gfCNCPoint2[12057] = {X 300.6818, Y 64.5076, Z -3.0000, A 0.000, B 0.000, C 0.000 }
gfCNCPoint2[12058] = {X 298.7202, Y 63.1248, Z -3.0000, A 0.000, B 0.000, C 0.000 }
gfCNCPoint2[12059] = {X 298.0340, Y 63.9594, Z -3.0000, A 0.000, B 0.000, C 0.000 }
gfCNCPoint2[12060] = {X 297.2321, Y 64.6835, Z -3.0000, A 0.000, B 0.000, C 0.000 }
gfCNCPoint2[12061] = {X 296.3321, Y 65.2812, Z -3.0000, A 0.000, B 0.000, C 0.000 }
gfCNCPoint2[12062] = {X 296.3321, Y 90.7168, Z -3.0000, A 0.000, B 0.000, C 0.000 }
gfCNCPoint2[12063] = {X 297.3123, Y 91.3793, Z -3.0000, A 0.000, B 0.000, C 0.000 }
gfCNCPoint2[12064] = {X 298.1728, Y 92.1913, Z -3.0000, A 0.000, B 0.000, C 0.000 }
gfCNCPoint2[12065] = {X 298.8912, Y 93.1314, Z -3.0000, A 0.000, B 0.000, C 0.000 }
gfCNCPoint2[12066] = {X 299.4485, Y 94.1751, Z -3.0000, A 0.000, B 0.000, C 0.000 }
gfCNCPoint2[12067] = {X 299.8302, Y 95.2950, Z -3.0000, A 0.000, B 0.000, C 0.000 }
gfCNCPoint2[12068] = {X 308.0994, Y 95.2950, Z -3.0000, A 0.000, B 0.000, C 0.000 }
gfCNCPoint2[12069] = {X 307.0963, Y 93.7116, Z -3.0000, A 0.000, B 0.000, C 0.000 }
gfCNCPoint2[12070] = {X 306.3004, Y 92.0147, Z -3.0000, A 0.000, B 0.000, C 0.000 }
gfCNCPoint2[12071] = {X 305.9924, Y 91.1576, Z -3.0000, A 0.000, B 0.000, C 0.000 }
gfCNCPoint2[12072] = {X 305.7375, Y 90.2832, Z -3.0000, A 0.000, B 0.000, C 0.000 }
gfCNCPoint2[12073] = {X 305.3413, Y 88.4127, Z -3.0000, A 0.000, B 0.000, C 0.000 }
gfCNCPoint2[12074] = {X 305.1069, Y 86.5150, Z -3.0000, A 0.000, B 0.000, C 0.000 }
gfCNCPoint2[12075] = {X 305.0361, Y 84.6043, Z -3.0000, A 0.000, B 0.000, C 0.000 }
gfCNCPoint2[12076] = {X 305.0373, Y 83.2289, Z -3.0000, A 0.000, B 0.000, C 0.000 }
gfCNCPoint2[12077] = {X 305.0373, Y 65.2849, Z -3.0000, A 0.000, B 0.000, C 0.000 }
gfCNCPoint2[12078] = {X 304.1350, Y 64.6870, Z -3.0000, A 0.000, B 0.000, C 0.000 }
gfCNCPoint2[12079] = {X 303.3314, Y 63.9619, Z -3.0000, A 0.000, B 0.000, C 0.000 }
gfCNCPoint2[12080] = {X 302.6441, Y 63.1258, Z -3.0000, A 0.000, B 0.000, C 0.000 }
gfCNCPoint2[12081] = {X 302.0791, Y 62.1784, Z -3.0000, A 0.000, B 0.000, C 0.000 }
gfCNCPoint2[12082] = {X 301.6638, Y 61.1566, Z -3.0000, A 0.000, B 0.000, C 0.000 }
gfCNCPoint2[12083] = {X 301.4076, Y 60.0837, Z -3.0000, A 0.000, B 0.000, C 0.000 }
gfCNCPoint2[12084] = {X 301.3164, Y 58.9845, Z -3.0000, A 0.000, B 0.000, C 0.000 }
gfCNCPoint2[12085] = {X 301.3162, Y 58.0000, Z -3.0000, A 0.000, B 0.000, C 0.000 }
gfCNCPoint2[12086] = {X 301.4018, Y 56.8868, Z -3.0000, A 0.000, B 0.000, C 0.000 }
gfCNCPoint2[12087] = {X 301.6567, Y 55.7997, Z -3.0000, A 0.000, B 0.000, C 0.000 }
gfCNCPoint2[12088] = {X 302.0747, Y 54.7645, Z -3.0000, A 0.000, B 0.000, C 0.000 }
gfCNCPoint2[12089] = {X 302.6462, Y 53.8053, Z -3.0000, A 0.000, B 0.000, C 0.000 }
gfCNCPoint2[12090] = {X 303.3281, Y 52.9755, Z -3.0000, A 0.000, B 0.000, C 0.000 }
gfCNCPoint2[12091] = {X 304.1247, Y 52.2551, Z -3.0000, A 0.000, B 0.000, C 0.000 }
gfCNCPoint2[12092] = {X 305.0187, Y 51.6597, Z -3.0000, A 0.000, B 0.000, C 0.000 }
gfCNCPoint2[12093] = {X 306.1514, Y 51.1428, Z -3.0000, A 0.000, B 0.000, C 0.000 }
gfCNCPoint2[12094] = {X 307.3557, Y 50.8265, Z -3.0000, A 0.000, B 0.000, C 0.000 }
gfCNCPoint2[12095] = {X 308.5962, Y 50.7200, Z -3.0000, A 0.000, B 0.000, C 0.000 }
gfCNCPoint2[12096] = {X 324.3107, Y 50.7200, Z -3.0000, A 0.000, B 0.000, C 0.000 }
gfCNCPoint2[12097] = {X 325.2469, Y 50.7804, Z -3.0000, A 0.000, B 0.000, C 0.000 }
gfCNCPoint2[12098] = {X 326.1675, Y 50.9608, Z -3.0000, A 0.000, B 0.000, C 0.000 }
gfCNCPoint2[12099] = {X 326.5260, Y 51.0653, Z -3.0000, A 0.000, B 0.000, C 0.000 }
gfCNCPoint2[12100] = {X 326.8787, Y 51.1880, Z -3.0000, A 0.000, B 0.000, C 0.000 }
gfCNCPoint2[12101] = {X 327.4520, Y 51.4326, Z -3.0000, A 0.000, B 0.000, C 0.000 }
gfCNCPoint2[12102] = {X 328.0023, Y 51.7254, Z -3.0000, A 0.000, B 0.000, C 0.000 }
gfCNCPoint2[12103] = {X 328.5421, Y 52.0760, Z -3.0000, A 0.000, B 0.000, C 0.000 }
gfCNCPoint2[12104] = {X 329.0488, Y 52.4729, Z -3.0000, A 0.000, B 0.000, C 0.000 }
gfCNCPoint2[12105] = {X 329.9268, Y 53.3678, Z -3.0000, A 0.000, B 0.000, C 0.000 }
gfCNCPoint2[12106] = {X 330.6383, Y 54.4000, Z -3.0000, A 0.000, B 0.000, C 0.000 }
gfCNCPoint2[12107] = {X 331.1621, Y 55.5390, Z -3.0000, A 0.000, B 0.000, C 0.000 }
gfCNCPoint2[12108] = {X 331.4827, Y 56.7510, Z -3.0000, A 0.000, B 0.000, C 0.000 }
gfCNCPoint2[12109] = {X 331.5907, Y 58.0000, Z -3.0000, A 0.000, B 0.000, C 0.000 }
gfCNCPoint2[12110] = {X 331.5907, Y 58.9400, Z -3.0000, A 0.000, B 0.000, C 0.000 }
gfCNCPoint2[12111] = {X 331.4731, Y 60.2169, Z -3.0000, A 0.000, B 0.000, C 0.000 }
gfCNCPoint2[12112] = {X 331.1345, Y 61.4536, Z -3.0000, A 0.000, B 0.000, C 0.000 }
gfCNCPoint2[12113] = {X 330.5852, Y 62.6123, Z -3.0000, A 0.000, B 0.000, C 0.000 }
gfCNCPoint2[12114] = {X 329.8422, Y 63.6573, Z -3.0000, A 0.000, B 0.000, C 0.000 }
gfCNCPoint2[12115] = {X 328.9282, Y 64.5567, Z -3.0000, A 0.000, B 0.000, C 0.000 }
gfCNCPoint2[12116] = {X 327.8712, Y 65.2827, Z -3.0000, A 0.000, B 0.000, C 0.000 }
gfCNCPoint2[12117] = {X 327.8726, Y 83.2150, Z -3.0000, A 0.000, B 0.000, C 0.000 }
gfCNCPoint2[12118] = {X 327.8860, Y 84.5922, Z -3.0000, A 0.000, B 0.000, C 0.000 }
gfCNCPoint2[12119] = {X 327.8954, Y 84.9546, Z -3.0000, A 0.000, B 0.000, C 0.000 }
gfCNCPoint2[12120] = {X 327.9223, Y 85.3160, Z -3.0000, A 0.000, B 0.000, C 0.000 }
gfCNCPoint2[12121] = {X 328.8635, Y 85.6736, Z -3.0000, A 0.000, B 0.000, C 0.000 }
gfCNCPoint2[12122] = {X 329.8331, Y 85.9449, Z -3.0000, A 0.000, B 0.000, C 0.000 }
gfCNCPoint2[12123] = {X 332.7072, Y 86.5208, Z -3.0000, A 0.000, B 0.000, C 0.000 }
gfCNCPoint2[12124] = {X 335.6155, Y 86.8875, Z -3.0000, A 0.000, B 0.000, C 0.000 }
gfCNCPoint2[12125] = {X 339.6624, Y 87.2011, Z -3.0000, A 0.000, B 0.000, C 0.000 }
gfCNCPoint2[12126] = {X 343.7177, Y 87.3767, Z -3.0000, A 0.000, B 0.000, C 0.000 }
gfCNCPoint2[12127] = {X 347.7766, Y 87.4140, Z -3.0000, A 0.000, B 0.000, C 0.000 }
gfCNCPoint2[12128] = {X 352.0642, Y 87.3773, Z -3.0000, A 0.000, B 0.000, C 0.000 }
gfCNCPoint2[12129] = {X 356.3477, Y 87.1860, Z -3.0000, A 0.000, B 0.000, C 0.000 }
gfCNCPoint2[12130] = {X 360.6216, Y 86.8405, Z -3.0000, A 0.000, B 0.000, C 0.000 }
gfCNCPoint2[12131] = {X 362.7646, Y 86.5743, Z -3.0000, A 0.000, B 0.000, C 0.000 }
gfCNCPoint2[12132] = {X 364.8876, Y 86.1795, Z -3.0000, A 0.000, B 0.000, C 0.000 }
gfCNCPoint2[12133] = {X 366.9831, Y 85.6575, Z -3.0000, A 0.000, B 0.000, C 0.000 }
gfCNCPoint2[12134] = {X 367.4432, Y 85.5111, Z -3.0000, A 0.000, B 0.000, C 0.000 }
gfCNCPoint2[12135] = {X 367.8895, Y 85.3269, Z -3.0000, A 0.000, B 0.000, C 0.000 }
gfCNCPoint2[12136] = {X 367.9430, Y 84.5784, Z -3.0000, A 0.000, B 0.000, C 0.000 }
gfCNCPoint2[12137] = {X 367.9608, Y 83.8282, Z -3.0000, A 0.000, B 0.000, C 0.000 }
gfCNCPoint2[12138] = {X 367.9593, Y 65.2843, Z -3.0000, A 0.000, B 0.000, C 0.000 }
gfCNCPoint2[12139] = {X 366.9053, Y 64.5652, Z -3.0000, A 0.000, B 0.000, C 0.000 }
gfCNCPoint2[12140] = {X 365.9931, Y 63.6732, Z -3.0000, A 0.000, B 0.000, C 0.000 }
gfCNCPoint2[12141] = {X 365.2505, Y 62.6356, Z -3.0000, A 0.000, B 0.000, C 0.000 }
gfCNCPoint2[12142] = {X 364.7006, Y 61.4843, Z -3.0000, A 0.000, B 0.000, C 0.000 }
gfCNCPoint2[12143] = {X 364.3601, Y 60.2547, Z -3.0000, A 0.000, B 0.000, C 0.000 }
gfCNCPoint2[12144] = {X 364.2395, Y 58.9845, Z -3.0000, A 0.000, B 0.000, C 0.000 }
gfCNCPoint2[12145] = {X 364.2393, Y 58.0000, Z -3.0000, A 0.000, B 0.000, C 0.000 }
gfCNCPoint2[12146] = {X 364.3499, Y 56.7358, Z -3.0000, A 0.000, B 0.000, C 0.000 }
gfCNCPoint2[12147] = {X 364.6783, Y 55.5101, Z -3.0000, A 0.000, B 0.000, C 0.000 }
gfCNCPoint2[12148] = {X 365.2146, Y 54.3600, Z -3.0000, A 0.000, B 0.000, C 0.000 }
gfCNCPoint2[12149] = {X 365.9425, Y 53.3205, Z -3.0000, A 0.000, B 0.000, C 0.000 }
gfCNCPoint2[12150] = {X 366.8398, Y 52.4232, Z -3.0000, A 0.000, B 0.000, C 0.000 }
gfCNCPoint2[12151] = {X 367.8793, Y 51.6953, Z -3.0000, A 0.000, B 0.000, C 0.000 }
gfCNCPoint2[12152] = {X 369.0294, Y 51.1590, Z -3.0000, A 0.000, B 0.000, C 0.000 }
gfCNCPoint2[12153] = {X 370.2551, Y 50.8306, Z -3.0000, A 0.000, B 0.000, C 0.000 }
gfCNCPoint2[12154] = {X 371.5193, Y 50.7200, Z -3.0000, A 0.000, B 0.000, C 0.000 }
gfCNCPoint2[12155] = {X 388.0597, Y 50.7200, Z -3.0000, A 0.000, B 0.000, C 0.000 }
gfCNCPoint2[12156] = {X 389.2271, Y 50.8142, Z -3.0000, A 0.000, B 0.000, C 0.000 }
gfCNCPoint2[12157] = {X 390.3643, Y 51.0944, Z -3.0000, A 0.000, B 0.000, C 0.000 }
gfCNCPoint2[12158] = {X 391.4418, Y 51.5533, Z -3.0000, A 0.000, B 0.000, C 0.000 }
gfCNCPoint2[12159] = {X 392.4319, Y 52.1791, Z -3.0000, A 0.000, B 0.000, C 0.000 }
gfCNCPoint2[12160] = {X 393.3087, Y 52.9556, Z -3.0000, A 0.000, B 0.000, C 0.000 }
gfCNCPoint2[12161] = {X 394.1855, Y 52.1791, Z -3.0000, A 0.000, B 0.000, C 0.000 }
gfCNCPoint2[12162] = {X 395.1756, Y 51.5533, Z -3.0000, A 0.000, B 0.000, C 0.000 }
gfCNCPoint2[12163] = {X 396.2531, Y 51.0944, Z -3.0000, A 0.000, B 0.000, C 0.000 }
gfCNCPoint2[12164] = {X 397.3903, Y 50.8142, Z -3.0000, A 0.000, B 0.000, C 0.000 }
gfCNCPoint2[12165] = {X 398.5577, Y 50.7200, Z -3.0000, A 0.000, B 0.000, C 0.000 }
gfCNCPoint2[12166] = {X 419.4886, Y 50.7200, Z -3.0000, A 0.000, B 0.000, C 0.000 }
gfCNCPoint2[12167] = {X 420.6740, Y 50.8172, Z -3.0000, A 0.000, B 0.000, C 0.000 }
gfCNCPoint2[12168] = {X 421.8278, Y 51.1060, Z -3.0000, A 0.000, B 0.000, C 0.000 }
gfCNCPoint2[12169] = {X 422.9191, Y 51.5790, Z -3.0000, A 0.000, B 0.000, C 0.000 }
gfCNCPoint2[12170] = {X 423.9189, Y 52.2233, Z -3.0000, A 0.000, B 0.000, C 0.000 }
gfCNCPoint2[12171] = {X 424.8004, Y 53.0217, Z -3.0000, A 0.000, B 0.000, C 0.000 }
gfCNCPoint2[12172] = {X 425.5401, Y 53.9531, Z -3.0000, A 0.000, B 0.000, C 0.000 }
gfCNCPoint2[12173] = {X 426.1183, Y 54.9925, Z -3.0000, A 0.000, B 0.000, C 0.000 }
gfCNCPoint2[12174] = {X 426.5196, Y 56.1122, Z -3.0000, A 0.000, B 0.000, C 0.000 }
gfCNCPoint2[12175] = {X 430.7007, Y 57.7417, Z -3.0000, A 0.000, B 0.000, C 0.000 }
gfCNCPoint2[12176] = {X 454.9001, Y 67.3428, Z -3.0000, A 0.000, B 0.000, C 0.000 }
gfCNCPoint2[12177] = {X 454.8999, Y 65.2844, Z -3.0000, A 0.000, B 0.000, C 0.000 }
gfCNCPoint2[12178] = {X 453.8924, Y 64.6032, Z -3.0000, A 0.000, B 0.000, C 0.000 }
gfCNCPoint2[12179] = {X 453.0124, Y 63.7638, Z -3.0000, A 0.000, B 0.000, C 0.000 }
gfCNCPoint2[12180] = {X 452.2844, Y 62.7896, Z -3.0000, A 0.000, B 0.000, C 0.000 }
gfCNCPoint2[12181] = {X 451.7287, Y 61.7078, Z -3.0000, A 0.000, B 0.000, C 0.000 }
gfCNCPoint2[12182] = {X 451.4297, Y 60.8260, Z -3.0000, A 0.000, B 0.000, C 0.000 }
gfCNCPoint2[12183] = {X 451.2457, Y 59.9132, Z -3.0000, A 0.000, B 0.000, C 0.000 }
gfCNCPoint2[12184] = {X 451.1798, Y 58.9845, Z -3.0000, A 0.000, B 0.000, C 0.000 }
gfCNCPoint2[12185] = {X 451.1796, Y 58.0000, Z -3.0000, A 0.000, B 0.000, C 0.000 }
gfCNCPoint2[12186] = {X 451.2795, Y 56.7981, Z -3.0000, A 0.000, B 0.000, C 0.000 }
gfCNCPoint2[12187] = {X 451.5765, Y 55.6291, Z -3.0000, A 0.000, B 0.000, C 0.000 }
gfCNCPoint2[12188] = {X 452.0624, Y 54.5253, Z -3.0000, A 0.000, B 0.000, C 0.000 }
gfCNCPoint2[12189] = {X 452.7238, Y 53.5168, Z -3.0000, A 0.000, B 0.000, C 0.000 }
gfCNCPoint2[12190] = {X 453.5427, Y 52.6313, Z -3.0000, A 0.000, B 0.000, C 0.000 }
gfCNCPoint2[12191] = {X 454.4966, Y 51.8932, Z -3.0000, A 0.000, B 0.000, C 0.000 }
gfCNCPoint2[12192] = {X 455.4133, Y 51.3880, Z -3.0000, A 0.000, B 0.000, C 0.000 }
gfCNCPoint2[12193] = {X 456.3931, Y 51.0195, Z -3.0000, A 0.000, B 0.000, C 0.000 }
gfCNCPoint2[12194] = {X 457.4155, Y 50.7953, Z -3.0000, A 0.000, B 0.000, C 0.000 }
gfCNCPoint2[12195] = {X 458.4596, Y 50.7200, Z -3.0000, A 0.000, B 0.000, C 0.000 }
gfCNCPoint2[12196] = {X 475.0000, Y 50.7200, Z -3.0000, A 0.000, B 0.000, C 0.000 }
gfCNCPoint2[12197] = {X 476.0441, Y 50.7953, Z -3.0000, A 0.000, B 0.000, C 0.000 }
gfCNCPoint2[12198] = {X 477.0665, Y 51.0195, Z -3.0000, A 0.000, B 0.000, C 0.000 }
gfCNCPoint2[12199] = {X 478.0463, Y 51.3880, Z -3.0000, A 0.000, B 0.000, C 0.000 }
gfCNCPoint2[12200] = {X 478.9630, Y 51.8932, Z -3.0000, A 0.000, B 0.000, C 0.000 }
gfCNCPoint2[12201] = {X 479.9169, Y 52.6313, Z -3.0000, A 0.000, B 0.000, C 0.000 }
gfCNCPoint2[12202] = {X 480.7358, Y 53.5168, Z -3.0000, A 0.000, B 0.000, C 0.000 }
gfCNCPoint2[12203] = {X 481.3972, Y 54.5253, Z -3.0000, A 0.000, B 0.000, C 0.000 }
gfCNCPoint2[12204] = {X 481.8831, Y 55.6291, Z -3.0000, A 0.000, B 0.000, C 0.000 }
gfCNCPoint2[12205] = {X 482.1801, Y 56.7981, Z -3.0000, A 0.000, B 0.000, C 0.000 }
gfCNCPoint2[12206] = {X 482.2800, Y 58.0000, Z -3.0000, A 0.000, B 0.000, C 0.000 }
gfCNCPoint2[12207] = {X 482.2798, Y 58.9942, Z -3.0000, A 0.000, B 0.000, C 0.000 }
gfCNCPoint2[12208] = {X 482.1577, Y 60.2627, Z -3.0000, A 0.000, B 0.000, C 0.000 }
gfCNCPoint2[12209] = {X 481.8164, Y 61.4904, Z -3.0000, A 0.000, B 0.000, C 0.000 }
gfCNCPoint2[12210] = {X 481.2662, Y 62.6399, Z -3.0000, A 0.000, B 0.000, C 0.000 }
gfCNCPoint2[12211] = {X 480.5240, Y 63.6758, Z -3.0000, A 0.000, B 0.000, C 0.000 }
gfCNCPoint2[12212] = {X 479.6125, Y 64.5664, Z -3.0000, A 0.000, B 0.000, C 0.000 }
gfCNCPoint2[12213] = {X 478.5597, Y 65.2844, Z -3.0000, A 0.000, B 0.000, C 0.000 }
gfCNCPoint2[12214] = {X 478.5601, Y 90.7248, Z -3.0000, A 0.000, B 0.000, C 0.000 }
gfCNCPoint2[12215] = {X 479.5426, Y 91.3833, Z -3.0000, A 0.000, B 0.000, C 0.000 }
gfCNCPoint2[12216] = {X 480.4051, Y 92.1928, Z -3.0000, A 0.000, B 0.000, C 0.000 }
gfCNCPoint2[12217] = {X 481.1245, Y 93.1317, Z -3.0000, A 0.000, B 0.000, C 0.000 }
gfCNCPoint2[12218] = {X 481.6818, Y 94.1750, Z -3.0000, A 0.000, B 0.000, C 0.000 }
gfCNCPoint2[12219] = {X 482.0621, Y 95.2950, Z -3.0000, A 0.000, B 0.000, C 0.000 }
gfCNCPoint2[12220] = {X 507.6818, Y 95.2950, Z -3.0000, A 0.000, B 0.000, C 0.000 }
gfCNCPoint2[12221] = {X 507.6818, Y 97.6950, Z -3.0000, A 0.000, B 0.000, C 0.000 }
gfCNCPoint2[12222] = {X 597.6965, Y 97.6950, Z -3.0000, A 0.000, B 0.000, C 0.000 }
gfCNCPoint2[12223] = {X 597.6965, Y 51.8000, Z -3.0000, A 0.000, B 0.000, C 0.000 }
gfCNCPoint2[12224] = {X 593.5565, Y 51.8000, Z -3.0000, A 0.000, B 0.000, C 0.000 }
gfCNCPoint2[12225] = {X 592.3428, Y 51.6908, Z -3.0000, A 0.000, B 0.000, C 0.000 }
gfCNCPoint2[12226] = {X 591.1680, Y 51.3667, Z -3.0000, A 0.000, B 0.000, C 0.000 }
gfCNCPoint2[12227] = {X 590.0699, Y 50.8381, Z -3.0000, A 0.000, B 0.000, C 0.000 }
gfCNCPoint2[12228] = {X 589.0838, Y 50.1220, Z -3.0000, A 0.000, B 0.000, C 0.000 }
gfCNCPoint2[12229] = {X 588.4736, Y 49.5171, Z -3.0000, A 0.000, B 0.000, C 0.000 }
gfCNCPoint2[12230] = {X 587.9446, Y 48.8401, Z -3.0000, A 0.000, B 0.000, C 0.000 }
gfCNCPoint2[12231] = {X 587.5052, Y 48.1018, Z -3.0000, A 0.000, B 0.000, C 0.000 }
gfCNCPoint2[12232] = {X 587.0658, Y 48.8401, Z -3.0000, A 0.000, B 0.000, C 0.000 }
gfCNCPoint2[12233] = {X 586.5368, Y 49.5171, Z -3.0000, A 0.000, B 0.000, C 0.000 }
gfCNCPoint2[12234] = {X 585.9266, Y 50.1220, Z -3.0000, A 0.000, B 0.000, C 0.000 }
gfCNCPoint2[12235] = {X 585.1803, Y 50.6880, Z -3.0000, A 0.000, B 0.000, C 0.000 }
gfCNCPoint2[12236] = {X 584.3634, Y 51.1461, Z -3.0000, A 0.000, B 0.000, C 0.000 }
gfCNCPoint2[12237] = {X 583.3013, Y 51.5442, Z -3.0000, A 0.000, B 0.000, C 0.000 }
gfCNCPoint2[12238] = {X 582.1877, Y 51.7603, Z -3.0000, A 0.000, B 0.000, C 0.000 }
gfCNCPoint2[12239] = {X 581.0538, Y 51.7882, Z -3.0000, A 0.000, B 0.000, C 0.000 }
gfCNCPoint2[12240] = {X 579.9310, Y 51.6273, Z -3.0000, A 0.000, B 0.000, C 0.000 }
gfCNCPoint2[12241] = {X 578.8505, Y 51.2819, Z -3.0000, A 0.000, B 0.000, C 0.000 }
gfCNCPoint2[12242] = {X 577.8425, Y 50.7618, Z -3.0000, A 0.000, B 0.000, C 0.000 }
gfCNCPoint2[12243] = {X 576.9350, Y 50.0813, Z -3.0000, A 0.000, B 0.000, C 0.000 }
gfCNCPoint2[12244] = {X 576.3133, Y 49.4513, Z -3.0000, A 0.000, B 0.000, C 0.000 }
gfCNCPoint2[12245] = {X 575.7786, Y 48.7459, Z -3.0000, A 0.000, B 0.000, C 0.000 }
gfCNCPoint2[12246] = {X 575.3401, Y 47.9770, Z -3.0000, A 0.000, B 0.000, C 0.000 }
gfCNCPoint2[12247] = {X 574.7637, Y 48.9470, Z -3.0000, A 0.000, B 0.000, C 0.000 }
gfCNCPoint2[12248] = {X 574.0348, Y 49.8083, Z -3.0000, A 0.000, B 0.000, C 0.000 }
gfCNCPoint2[12249] = {X 573.8920, Y 49.9470, Z -3.0000, A 0.000, B 0.000, C 0.000 }
gfCNCPoint2[12250] = {X 573.7453, Y 50.0813, Z -3.0000, A 0.000, B 0.000, C 0.000 }
gfCNCPoint2[12251] = {X 572.7526, Y 50.8143, Z -3.0000, A 0.000, B 0.000, C 0.000 }
gfCNCPoint2[12252] = {X 571.6437, Y 51.3558, Z -3.0000, A 0.000, B 0.000, C 0.000 }
gfCNCPoint2[12253] = {X 570.4553, Y 51.6880, Z -3.0000, A 0.000, B 0.000, C 0.000 }
gfCNCPoint2[12254] = {X 569.2264, Y 51.8000, Z -3.0000, A 0.000, B 0.000, C 0.000 }
gfCNCPoint2[12255] = {X 562.4443, Y 51.8000, Z -3.0000, A 0.000, B 0.000, C 0.000 }
gfCNCPoint2[12256] = {X 561.2635, Y 51.6967, Z -3.0000, A 0.000, B 0.000, C 0.000 }
gfCNCPoint2[12257] = {X 560.1186, Y 51.3899, Z -3.0000, A 0.000, B 0.000, C 0.000 }
gfCNCPoint2[12258] = {X 559.0443, Y 50.8890, Z -3.0000, A 0.000, B 0.000, C 0.000 }
gfCNCPoint2[12259] = {X 558.0733, Y 50.2091, Z -3.0000, A 0.000, B 0.000, C 0.000 }
gfCNCPoint2[12260] = {X 557.2352, Y 49.3710, Z -3.0000, A 0.000, B 0.000, C 0.000 }
gfCNCPoint2[12261] = {X 556.5553, Y 48.4000, Z -3.0000, A 0.000, B 0.000, C 0.000 }
gfCNCPoint2[12262] = {X 556.0544, Y 47.3257, Z -3.0000, A 0.000, B 0.000, C 0.000 }
gfCNCPoint2[12263] = {X 555.7476, Y 46.1808, Z -3.0000, A 0.000, B 0.000, C 0.000 }
gfCNCPoint2[12264] = {X 555.6443, Y 45.0000, Z -3.0000, A 0.000, B 0.000, C 0.000 }
gfCNCPoint2[12265] = {X 555.6443, Y 44.0663, Z -3.0000, A 0.000, B 0.000, C 0.000 }
gfCNCPoint2[12266] = {X 555.7457, Y 42.9115, Z -3.0000, A 0.000, B 0.000, C 0.000 }
gfCNCPoint2[12267] = {X 556.0407, Y 41.7905, Z -3.0000, A 0.000, B 0.000, C 0.000 }
gfCNCPoint2[12268] = {X 556.5208, Y 40.7354, Z -3.0000, A 0.000, B 0.000, C 0.000 }
gfCNCPoint2[12269] = {X 557.1724, Y 39.7767, Z -3.0000, A 0.000, B 0.000, C 0.000 }
gfCNCPoint2[12270] = {X 557.1724, Y 10.2290, Z -3.0000, A 0.000, B 0.000, C 0.000 }
gfCNCPoint2[12271] = {X 556.5260, Y 9.2828, Z -3.0000, A 0.000, B 0.000, C 0.000 }
gfCNCPoint2[12272] = {X 556.0477, Y 8.2414, Z -3.0000, A 0.000, B 0.000, C 0.000 }
gfCNCPoint2[12273] = {X 555.7511, Y 7.1345, Z -3.0000, A 0.000, B 0.000, C 0.000 }
gfCNCPoint2[12274] = {X 555.6446, Y 5.9935, Z -3.0000, A 0.000, B 0.000, C 0.000 }
gfCNCPoint2[12275] = {X 555.6443, Y 5.0000, Z -3.0000, A 0.000, B 0.000, C 0.000 }
gfCNCPoint2[12276] = {X 555.6452, Y 4.8910, Z -3.0000, A 0.000, B 0.000, C 0.000 }
gfCNCPoint2[12277] = {X 555.6478, Y 4.7820, Z -3.0000, A 0.000, B 0.000, C 0.000 }
gfCNCPoint2[12278] = {X 555.8079, Y 3.5175, Z -3.0000, A 0.000, B 0.000, C 0.000 }
gfCNCPoint2[12279] = {X 556.2011, Y 2.3050, Z -3.0000, A 0.000, B 0.000, C 0.000 }
gfCNCPoint2[12280] = {X 358.2581, Y 2.3050, Z -3.0000, A 0.000, B 0.000, C 0.000 }
gfCNCPoint2[12281] = {X 360.1196, Y 3.4747, Z -3.0000, A 0.000, B 0.000, C 0.000 }
gfCNCPoint2[12282] = {X 361.8525, Y 4.8276, Z -3.0000, A 0.000, B 0.000, C 0.000 }
gfCNCPoint2[12283] = {X 363.4387, Y 6.3498, Z -3.0000, A 0.000, B 0.000, C 0.000 }
gfCNCPoint2[12284] = {X 363.7843, Y 6.7258, Z -3.0000, A 0.000, B 0.000, C 0.000 }
gfCNCPoint2[12285] = {X 364.1208, Y 7.1099, Z -3.0000, A 0.000, B 0.000, C 0.000 }
gfCNCPoint2[12286] = {X 365.6213, Y 9.0462, Z -3.0000, A 0.000, B 0.000, C 0.000 }
gfCNCPoint2[12287] = {X 366.9272, Y 11.1187, Z -3.0000, A 0.000, B 0.000, C 0.000 }
gfCNCPoint2[12288] = {X 368.0265, Y 13.3079, Z -3.0000, A 0.000, B 0.000, C 0.000 }
gfCNCPoint2[12289] = {X 368.9087, Y 15.5932, Z -3.0000, A 0.000, B 0.000, C 0.000 }
gfCNCPoint2[12290] = {X 369.5655, Y 17.9532, Z -3.0000, A 0.000, B 0.000, C 0.000 }
gfCNCPoint2[12291] = {X 370.0551, Y 20.6344, Z -3.0000, A 0.000, B 0.000, C 0.000 }
gfCNCPoint2[12292] = {X 370.3162, Y 23.3475, Z -3.0000, A 0.000, B 0.000, C 0.000 }
gfCNCPoint2[12293] = {X 370.3467, Y 26.0729, Z -3.0000, A 0.000, B 0.000, C 0.000 }
gfCNCPoint2[12294] = {X 370.1465, Y 28.7912, Z -3.0000, A 0.000, B 0.000, C 0.000 }
gfCNCPoint2[12295] = {X 369.7171, Y 31.4827, Z -3.0000, A 0.000, B 0.000, C 0.000 }
gfCNCPoint2[12296] = {X 369.1813, Y 33.6350, Z -3.0000, A 0.000, B 0.000, C 0.000 }
gfCNCPoint2[12297] = {X 368.4574, Y 35.7315, Z -3.0000, A 0.000, B 0.000, C 0.000 }
gfCNCPoint2[12298] = {X 367.5511, Y 37.7559, Z -3.0000, A 0.000, B 0.000, C 0.000 }
gfCNCPoint2[12299] = {X 366.4695, Y 39.6923, Z -3.0000, A 0.000, B 0.000, C 0.000 }
gfCNCPoint2[12300] = {X 365.2210, Y 41.5255, Z -3.0000, A 0.000, B 0.000, C 0.000 }
gfCNCPoint2[12301] = {X 363.9635, Y 43.0750, Z -3.0000, A 0.000, B 0.000, C 0.000 }
gfCNCPoint2[12302] = {X 362.5750, Y 44.5082, Z -3.0000, A 0.000, B 0.000, C 0.000 }
gfCNCPoint2[12303] = {X 361.0663, Y 45.8143, Z -3.0000, A 0.000, B 0.000, C 0.000 }
gfCNCPoint2[12304] = {X 359.4488, Y 46.9830, Z -3.0000, A 0.000, B 0.000, C 0.000 }
gfCNCPoint2[12305] = {X 357.7352, Y 48.0055, Z -3.0000, A 0.000, B 0.000, C 0.000 }
gfCNCPoint2[12306] = {X 355.7254, Y 48.9198, Z -3.0000, A 0.000, B 0.000, C 0.000 }
gfCNCPoint2[12307] = {X 353.6378, Y 49.6388, Z -3.0000, A 0.000, B 0.000, C 0.000 }
gfCNCPoint2[12308] = {X 351.4913, Y 50.1561, Z -3.0000, A 0.000, B 0.000, C 0.000 }
gfCNCPoint2[12309] = {X 349.3053, Y 50.4668, Z -3.0000, A 0.000, B 0.000, C 0.000 }
gfCNCPoint2[12310] = {X 347.0997, Y 50.5683, Z -3.0000, A 0.000, B 0.000, C 0.000 }
gfCNCPoint2[12311] = {X 344.9865, Y 50.5320, Z -3.0000, A 0.000, B 0.000, C 0.000 }
gfCNCPoint2[12312] = {X 342.8843, Y 50.3128, Z -3.0000, A 0.000, B 0.000, C 0.000 }
gfCNCPoint2[12313] = {X 340.8090, Y 49.9122, Z -3.0000, A 0.000, B 0.000, C 0.000 }
gfCNCPoint2[12314] = {X 338.7763, Y 49.3332, Z -3.0000, A 0.000, B 0.000, C 0.000 }
gfCNCPoint2[12315] = {X 336.8014, Y 48.5803, Z -3.0000, A 0.000, B 0.000, C 0.000 }
gfCNCPoint2[12316] = {X 334.8991, Y 47.6591, Z -3.0000, A 0.000, B 0.000, C 0.000 }
gfCNCPoint2[12317] = {X 333.3420, Y 46.7029, Z -3.0000, A 0.000, B 0.000, C 0.000 }
gfCNCPoint2[12318] = {X 331.8608, Y 45.6328, Z -3.0000, A 0.000, B 0.000, C 0.000 }
gfCNCPoint2[12319] = {X 330.4638, Y 44.4550, Z -3.0000, A 0.000, B 0.000, C 0.000 }
gfCNCPoint2[12320] = {X 329.4666, Y 44.4079, Z -3.0000, A 0.000, B 0.000, C 0.000 }
gfCNCPoint2[12321] = {X 328.4997, Y 44.1588, Z -3.0000, A 0.000, B 0.000, C 0.000 }
gfCNCPoint2[12322] = {X 327.6038, Y 43.7181, Z -3.0000, A 0.000, B 0.000, C 0.000 }
gfCNCPoint2[12323] = {X 326.8164, Y 43.1044, Z -3.0000, A 0.000, B 0.000, C 0.000 }
gfCNCPoint2[12324] = {X 326.1897, Y 42.4934, Z -3.0000, A 0.000, B 0.000, C 0.000 }
gfCNCPoint2[12325] = {X 325.5686, Y 41.7541, Z -3.0000, A 0.000, B 0.000, C 0.000 }
gfCNCPoint2[12326] = {X 325.1052, Y 40.9070, Z -3.0000, A 0.000, B 0.000, C 0.000 }
gfCNCPoint2[12327] = {X 324.8177, Y 39.9852, Z -3.0000, A 0.000, B 0.000, C 0.000 }
gfCNCPoint2[12328] = {X 324.7172, Y 39.0249, Z -3.0000, A 0.000, B 0.000, C 0.000 }
gfCNCPoint2[12329] = {X 324.8079, Y 38.0635, Z -3.0000, A 0.000, B 0.000, C 0.000 }
gfCNCPoint2[12330] = {X 325.0860, Y 37.1389, Z -3.0000, A 0.000, B 0.000, C 0.000 }
gfCNCPoint2[12331] = {X 325.5408, Y 36.2871, Z -3.0000, A 0.000, B 0.000, C 0.000 }
gfCNCPoint2[12332] = {X 329.7739, Y 29.9576, Z -3.0000, A 0.000, B 0.000, C 0.000 }
gfCNCPoint2[12333] = {X 330.4584, Y 29.1427, Z -3.0000, A 0.000, B 0.000, C 0.000 }
gfCNCPoint2[12334] = {X 331.3033, Y 28.4956, Z -3.0000, A 0.000, B 0.000, C 0.000 }
gfCNCPoint2[12335] = {X 332.2684, Y 28.0471, Z -3.0000, A 0.000, B 0.000, C 0.000 }
gfCNCPoint2[12336] = {X 333.3078, Y 27.8184, Z -3.0000, A 0.000, B 0.000, C 0.000 }
gfCNCPoint2[12337] = {X 334.3720, Y 27.8205, Z -3.0000, A 0.000, B 0.000, C 0.000 }
gfCNCPoint2[12338] = {X 335.4105, Y 28.0532, Z -3.0000, A 0.000, B 0.000, C 0.000 }
gfCNCPoint2[12339] = {X 336.3738, Y 28.5055, Z -3.0000, A 0.000, B 0.000, C 0.000 }
gfCNCPoint2[12340] = {X 337.2162, Y 29.1559, Z -3.0000, A 0.000, B 0.000, C 0.000 }
gfCNCPoint2[12341] = {X 337.7864, Y 29.7052, Z -3.0000, A 0.000, B 0.000, C 0.000 }
gfCNCPoint2[12342] = {X 338.3565, Y 30.3621, Z -3.0000, A 0.000, B 0.000, C 0.000 }
gfCNCPoint2[12343] = {X 338.8010, Y 31.1097, Z -3.0000, A 0.000, B 0.000, C 0.000 }
gfCNCPoint2[12344] = {X 339.1058, Y 31.9245, Z -3.0000, A 0.000, B 0.000, C 0.000 }
gfCNCPoint2[12345] = {X 339.2610, Y 32.7803, Z -3.0000, A 0.000, B 0.000, C 0.000 }
gfCNCPoint2[12346] = {X 339.2618, Y 33.6502, Z -3.0000, A 0.000, B 0.000, C 0.000 }
gfCNCPoint2[12347] = {X 339.9062, Y 34.2217, Z -3.0000, A 0.000, B 0.000, C 0.000 }
gfCNCPoint2[12348] = {X 340.5750, Y 34.7645, Z -3.0000, A 0.000, B 0.000, C 0.000 }
gfCNCPoint2[12349] = {X 341.8068, Y 35.5732, Z -3.0000, A 0.000, B 0.000, C 0.000 }
gfCNCPoint2[12350] = {X 343.1435, Y 36.1931, Z -3.0000, A 0.000, B 0.000, C 0.000 }
gfCNCPoint2[12351] = {X 344.5565, Y 36.6111, Z -3.0000, A 0.000, B 0.000, C 0.000 }
gfCNCPoint2[12352] = {X 346.0154, Y 36.8180, Z -3.0000, A 0.000, B 0.000, C 0.000 }
gfCNCPoint2[12353] = {X 347.4889, Y 36.8096, Z -3.0000, A 0.000, B 0.000, C 0.000 }
gfCNCPoint2[12354] = {X 348.8381, Y 36.6284, Z -3.0000, A 0.000, B 0.000, C 0.000 }
gfCNCPoint2[12355] = {X 350.1399, Y 36.2301, Z -3.0000, A 0.000, B 0.000, C 0.000 }
gfCNCPoint2[12356] = {X 351.3595, Y 35.6252, Z -3.0000, A 0.000, B 0.000, C 0.000 }
gfCNCPoint2[12357] = {X 352.4644, Y 34.8298, Z -3.0000, A 0.000, B 0.000, C 0.000 }
gfCNCPoint2[12358] = {X 353.5661, Y 33.7599, Z -3.0000, A 0.000, B 0.000, C 0.000 }
gfCNCPoint2[12359] = {X 354.5195, Y 32.5561, Z -3.0000, A 0.000, B 0.000, C 0.000 }
gfCNCPoint2[12360] = {X 355.3086, Y 31.2387, Z -3.0000, A 0.000, B 0.000, C 0.000 }
gfCNCPoint2[12361] = {X 355.9199, Y 29.8299, Z -3.0000, A 0.000, B 0.000, C 0.000 }
gfCNCPoint2[12362] = {X 356.3432, Y 28.3538, Z -3.0000, A 0.000, B 0.000, C 0.000 }
gfCNCPoint2[12363] = {X 356.6078, Y 26.7186, Z -3.0000, A 0.000, B 0.000, C 0.000 }
gfCNCPoint2[12364] = {X 356.7155, Y 25.0657, Z -3.0000, A 0.000, B 0.000, C 0.000 }
gfCNCPoint2[12365] = {X 356.6654, Y 23.4100, Z -3.0000, A 0.000, B 0.000, C 0.000 }
gfCNCPoint2[12366] = {X 356.4579, Y 21.7667, Z -3.0000, A 0.000, B 0.000, C 0.000 }
gfCNCPoint2[12367] = {X 356.1376, Y 20.3836, Z -3.0000, A 0.000, B 0.000, C 0.000 }
gfCNCPoint2[12368] = {X 355.6485, Y 19.0509, Z -3.0000, A 0.000, B 0.000, C 0.000 }
gfCNCPoint2[12369] = {X 354.9980, Y 17.7891, Z -3.0000, A 0.000, B 0.000, C 0.000 }
gfCNCPoint2[12370] = {X 354.1962, Y 16.6175, Z -3.0000, A 0.000, B 0.000, C 0.000 }
gfCNCPoint2[12371] = {X 353.3641, Y 15.6890, Z -3.0000, A 0.000, B 0.000, C 0.000 }
gfCNCPoint2[12372] = {X 352.4075, Y 14.8894, Z -3.0000, A 0.000, B 0.000, C 0.000 }
gfCNCPoint2[12373] = {X 351.3462, Y 14.2351, Z -3.0000, A 0.000, B 0.000, C 0.000 }
gfCNCPoint2[12374] = {X 350.2021, Y 13.7396, Z -3.0000, A 0.000, B 0.000, C 0.000 }
gfCNCPoint2[12375] = {X 348.9988, Y 13.4131, Z -3.0000, A 0.000, B 0.000, C 0.000 }
gfCNCPoint2[12376] = {X 347.3615, Y 13.2064, Z -3.0000, A 0.000, B 0.000, C 0.000 }
gfCNCPoint2[12377] = {X 345.7113, Y 13.2118, Z -3.0000, A 0.000, B 0.000, C 0.000 }
gfCNCPoint2[12378] = {X 344.0754, Y 13.4290, Z -3.0000, A 0.000, B 0.000, C 0.000 }
gfCNCPoint2[12379] = {X 342.4810, Y 13.8545, Z -3.0000, A 0.000, B 0.000, C 0.000 }
gfCNCPoint2[12380] = {X 340.9544, Y 14.4812, Z -3.0000, A 0.000, B 0.000, C 0.000 }
gfCNCPoint2[12381] = {X 339.5210, Y 15.2988, Z -3.0000, A 0.000, B 0.000, C 0.000 }
gfCNCPoint2[12382] = {X 339.4273, Y 16.1847, Z -3.0000, A 0.000, B 0.000, C 0.000 }
gfCNCPoint2[12383] = {X 339.1742, Y 17.0388, Z -3.0000, A 0.000, B 0.000, C 0.000 }
gfCNCPoint2[12384] = {X 338.7700, Y 17.8326, Z -3.0000, A 0.000, B 0.000, C 0.000 }
gfCNCPoint2[12385] = {X 338.2282, Y 18.5397, Z -3.0000, A 0.000, B 0.000, C 0.000 }
gfCNCPoint2[12386] = {X 337.5670, Y 19.1366, Z -3.0000, A 0.000, B 0.000, C 0.000 }
gfCNCPoint2[12387] = {X 336.8400, Y 19.6716, Z -3.0000, A 0.000, B 0.000, C 0.000 }
gfCNCPoint2[12388] = {X 335.9171, Y 20.1909, Z -3.0000, A 0.000, B 0.000, C 0.000 }
gfCNCPoint2[12389] = {X 334.9039, Y 20.4988, Z -3.0000, A 0.000, B 0.000, C 0.000 }
gfCNCPoint2[12390] = {X 333.8481, Y 20.5809, Z -3.0000, A 0.000, B 0.000, C 0.000 }
gfCNCPoint2[12391] = {X 332.7995, Y 20.4334, Z -3.0000, A 0.000, B 0.000, C 0.000 }
gfCNCPoint2[12392] = {X 331.8074, Y 20.0631, Z -3.0000, A 0.000, B 0.000, C 0.000 }
gfCNCPoint2[12393] = {X 330.9186, Y 19.4875, Z -3.0000, A 0.000, B 0.000, C 0.000 }
gfCNCPoint2[12394] = {X 330.1748, Y 18.7338, Z -3.0000, A 0.000, B 0.000, C 0.000 }
gfCNCPoint2[12395] = {X 329.6111, Y 17.8373, Z -3.0000, A 0.000, B 0.000, C 0.000 }
gfCNCPoint2[12396] = {X 326.0906, Y 10.5950, Z -3.0000, A 0.000, B 0.000, C 0.000 }
gfCNCPoint2[12397] = {X 325.7555, Y 9.6856, Z -3.0000, A 0.000, B 0.000, C 0.000 }
gfCNCPoint2[12398] = {X 325.6067, Y 8.7279, Z -3.0000, A 0.000, B 0.000, C 0.000 }
gfCNCPoint2[12399] = {X 325.6502, Y 7.7597, Z -3.0000, A 0.000, B 0.000, C 0.000 }
gfCNCPoint2[12400] = {X 325.8841, Y 6.8192, Z -3.0000, A 0.000, B 0.000, C 0.000 }
gfCNCPoint2[12401] = {X 326.2993, Y 5.9434, Z -3.0000, A 0.000, B 0.000, C 0.000 }
gfCNCPoint2[12402] = {X 326.9295, Y 5.1131, Z -3.0000, A 0.000, B 0.000, C 0.000 }
gfCNCPoint2[12403] = {X 327.7216, Y 4.4356, Z -3.0000, A 0.000, B 0.000, C 0.000 }
gfCNCPoint2[12404] = {X 328.3968, Y 3.9733, Z -3.0000, A 0.000, B 0.000, C 0.000 }
gfCNCPoint2[12405] = {X 329.3296, Y 3.4827, Z -3.0000, A 0.000, B 0.000, C 0.000 }
gfCNCPoint2[12406] = {X 330.3460, Y 3.2039, Z -3.0000, A 0.000, B 0.000, C 0.000 }
gfCNCPoint2[12407] = {X 331.3986, Y 3.1499, Z -3.0000, A 0.000, B 0.000, C 0.000 }
gfCNCPoint2[12408] = {X 332.4382, Y 3.3231, Z -3.0000, A 0.000, B 0.000, C 0.000 }
gfCNCPoint2[12409] = {X 333.3757, Y 2.7964, Z -3.0000, A 0.000, B 0.000, C 0.000 }
gfCNCPoint2[12410] = {X 334.3322, Y 2.3050, Z -3.0000, A 0.000, B 0.000, C 0.000 }
gfCNCPoint2[12411] = {X 334.5436, Y 2.7360, Z -3.0000, A 0.000, B 0.000, C 0.000 }
gfCNCPoint2[12412] = {X 335.0198, Y 2.5079, Z -3.0000, A 0.000, B 0.000, C 0.000 }
gfCNCPoint2[12413] = {X 335.5002, Y 2.2886, Z -3.0000, A 0.000, B 0.000, C 0.000 }
gfCNCPoint2[12414] = {X 335.8480, Y 2.1338, Z -3.0000, A 0.000, B 0.000, C 0.000 }
gfCNCPoint2[12415] = {X 337.9511, Y 1.3133, Z -3.0000, A 0.000, B 0.000, C 0.000 }
gfCNCPoint2[12416] = {X 340.1168, Y 0.6758, Z -3.0000, A 0.000, B 0.000, C 0.000 }
gfCNCPoint2[12417] = {X 342.3290, Y 0.2258, Z -3.0000, A 0.000, B 0.000, C 0.000 }
gfCNCPoint2[12418] = {X 344.5717, Y -0.0331, Z -3.0000, A 0.000, B 0.000, C 0.000 }
gfCNCPoint2[12419] = {X 346.8283, Y -0.0993, Z -3.0000, A 0.000, B 0.000, C 0.000 }
gfCNCPoint2[12420] = {X 349.0822, Y 0.0279, Z -3.0000, A 0.000, B 0.000, C 0.000 }
gfCNCPoint2[12421] = {X 351.3170, Y 0.3475, Z -3.0000, A 0.000, B 0.000, C 0.000 }
gfCNCPoint2[12422] = {X 351.8874, Y 0.4533, Z -3.0000, A 0.000, B 0.000, C 0.000 }
gfCNCPoint2[12423] = {X 353.8291, Y 0.9413, Z -3.0000, A 0.000, B 0.000, C 0.000 }
gfCNCPoint2[12424] = {X 355.7158, Y 1.6110, Z -3.0000, A 0.000, B 0.000, C 0.000 }
gfCNCPoint2[12425] = {X 357.5305, Y 2.4566, Z -3.0000, A 0.000, B 0.000, C 0.000 }
gfCNCPoint2[12426] = {X 359.2570, Y 3.4702, Z -3.0000, A 0.000, B 0.000, C 0.000 }
gfCNCPoint2[12427] = {X 360.8796, Y 4.6429, Z -3.0000, A 0.000, B 0.000, C 0.000 }
gfCNCPoint2[12428] = {X 362.3838, Y 5.9641, Z -3.0000, A 0.000, B 0.000, C 0.000 }
gfCNCPoint2[12429] = {X 363.7561, Y 7.4219, Z -3.0000, A 0.000, B 0.000, C 0.000 }
gfCNCPoint2[12430] = {X 365.2280, Y 9.3215, Z -3.0000, A 0.000, B 0.000, C 0.000 }
gfCNCPoint2[12431] = {X 366.5092, Y 11.3547, Z -3.0000, A 0.000, B 0.000, C 0.000 }
gfCNCPoint2[12432] = {X 367.5876, Y 13.5023, Z -3.0000, A 0.000, B 0.000, C 0.000 }
gfCNCPoint2[12433] = {X 368.4530, Y 15.7442, Z -3.0000, A 0.000, B 0.000, C 0.000 }
gfCNCPoint2[12434] = {X 369.0974, Y 18.0593, Z -3.0000, A 0.000, B 0.000, C 0.000 }
gfCNCPoint2[12435] = {X 369.5797, Y 20.7006, Z -3.0000, A 0.000, B 0.000, C 0.000 }
gfCNCPoint2[12436] = {X 369.8369, Y 23.3732, Z -3.0000, A 0.000, B 0.000, C 0.000 }
gfCNCPoint2[12437] = {X 369.8669, Y 26.0580, Z -3.0000, A 0.000, B 0.000, C 0.000 }
gfCNCPoint2[12438] = {X 369.6698, Y 28.7357, Z -3.0000, A 0.000, B 0.000, C 0.000 }
gfCNCPoint2[12439] = {X 369.2467, Y 31.3871, Z -3.0000, A 0.000, B 0.000, C 0.000 }
gfCNCPoint2[12440] = {X 368.7211, Y 33.4985, Z -3.0000, A 0.000, B 0.000, C 0.000 }
gfCNCPoint2[12441] = {X 368.0110, Y 35.5551, Z -3.0000, A 0.000, B 0.000, C 0.000 }
gfCNCPoint2[12442] = {X 367.1219, Y 37.5409, Z -3.0000, A 0.000, B 0.000, C 0.000 }
gfCNCPoint2[12443] = {X 366.0608, Y 39.4405, Z -3.0000, A 0.000, B 0.000, C 0.000 }
gfCNCPoint2[12444] = {X 364.8361, Y 41.2388, Z -3.0000, A 0.000, B 0.000, C 0.000 }
gfCNCPoint2[12445] = {X 363.6039, Y 42.7570, Z -3.0000, A 0.000, B 0.000, C 0.000 }
gfCNCPoint2[12446] = {X 362.2434, Y 44.1612, Z -3.0000, A 0.000, B 0.000, C 0.000 }
gfCNCPoint2[12447] = {X 360.7649, Y 45.4406, Z -3.0000, A 0.000, B 0.000, C 0.000 }
gfCNCPoint2[12448] = {X 359.1798, Y 46.5854, Z -3.0000, A 0.000, B 0.000, C 0.000 }
gfCNCPoint2[12449] = {X 357.5004, Y 47.5867, Z -3.0000, A 0.000, B 0.000, C 0.000 }
gfCNCPoint2[12450] = {X 355.5335, Y 48.4797, Z -3.0000, A 0.000, B 0.000, C 0.000 }
gfCNCPoint2[12451] = {X 353.4907, Y 49.1818, Z -3.0000, A 0.000, B 0.000, C 0.000 }
gfCNCPoint2[12452] = {X 351.3904, Y 49.6867, Z -3.0000, A 0.000, B 0.000, C 0.000 }
gfCNCPoint2[12453] = {X 349.2517, Y 49.9898, Z -3.0000, A 0.000, B 0.000, C 0.000 }
gfCNCPoint2[12454] = {X 347.0938, Y 50.0883, Z -3.0000, A 0.000, B 0.000, C 0.000 }
gfCNCPoint2[12455] = {X 345.0198, Y 50.0531, Z -3.0000, A 0.000, B 0.000, C 0.000 }
gfCNCPoint2[12456] = {X 342.9566, Y 49.8382, Z -3.0000, A 0.000, B 0.000, C 0.000 }
gfCNCPoint2[12457] = {X 340.9198, Y 49.4451, Z -3.0000, A 0.000, B 0.000, C 0.000 }
gfCNCPoint2[12458] = {X 338.9248, Y 48.8767, Z -3.0000, A 0.000, B 0.000, C 0.000 }
gfCNCPoint2[12459] = {X 336.9867, Y 48.1375, Z -3.0000, A 0.000, B 0.000, C 0.000 }
gfCNCPoint2[12460] = {X 335.1200, Y 47.2328, Z -3.0000, A 0.000, B 0.000, C 0.000 }
gfCNCPoint2[12461] = {X 333.5417, Y 46.2591, Z -3.0000, A 0.000, B 0.000, C 0.000 }
gfCNCPoint2[12462] = {X 332.0436, Y 45.1661, Z -3.0000, A 0.000, B 0.000, C 0.000 }
gfCNCPoint2[12463] = {X 330.6347, Y 43.9603, Z -3.0000, A 0.000, B 0.000, C 0.000 }
gfCNCPoint2[12464] = {X 329.6761, Y 43.9518, Z -3.0000, A 0.000, B 0.000, C 0.000 }
gfCNCPoint2[12465] = {X 328.7421, Y 43.7359, Z -3.0000, A 0.000, B 0.000, C 0.000 }
gfCNCPoint2[12466] = {X 327.8770, Y 43.3228, Z -3.0000, A 0.000, B 0.000, C 0.000 }
gfCNCPoint2[12467] = {X 327.1219, Y 42.7321, Z -3.0000, A 0.000, B 0.000, C 0.000 }
gfCNCPoint2[12468] = {X 326.5249, Y 42.1498, Z -3.0000, A 0.000, B 0.000, C 0.000 }
gfCNCPoint2[12469] = {X 325.8848, Y 41.3619, Z -3.0000, A 0.000, B 0.000, C 0.000 }
gfCNCPoint2[12470] = {X 325.4424, Y 40.4483, Z -3.0000, A 0.000, B 0.000, C 0.000 }
gfCNCPoint2[12471] = {X 325.2210, Y 39.4576, Z -3.0000, A 0.000, B 0.000, C 0.000 }
gfCNCPoint2[12472] = {X 325.2326, Y 38.4426, Z -3.0000, A 0.000, B 0.000, C 0.000 }
gfCNCPoint2[12473] = {X 325.4765, Y 37.4572, Z -3.0000, A 0.000, B 0.000, C 0.000 }
gfCNCPoint2[12474] = {X 325.9397, Y 36.5539, Z -3.0000, A 0.000, B 0.000, C 0.000 }
gfCNCPoint2[12475] = {X 330.1988, Y 30.1861, Z -3.0000, A 0.000, B 0.000, C 0.000 }
gfCNCPoint2[12476] = {X 330.8195, Y 29.4619, Z -3.0000, A 0.000, B 0.000, C 0.000 }
gfCNCPoint2[12477] = {X 331.5816, Y 28.8884, Z -3.0000, A 0.000, B 0.000, C 0.000 }
gfCNCPoint2[12478] = {X 332.4495, Y 28.4927, Z -3.0000, A 0.000, B 0.000, C 0.000 }
gfCNCPoint2[12479] = {X 333.3822, Y 28.2932, Z -3.0000, A 0.000, B 0.000, C 0.000 }
gfCNCPoint2[12480] = {X 334.3360, Y 28.2995, Z -3.0000, A 0.000, B 0.000, C 0.000 }
gfCNCPoint2[12481] = {X 335.2660, Y 28.5111, Z -3.0000, A 0.000, B 0.000, C 0.000 }
gfCNCPoint2[12482] = {X 336.1286, Y 28.9182, Z -3.0000, A 0.000, B 0.000, C 0.000 }
gfCNCPoint2[12483] = {X 336.8832, Y 29.5016, Z -3.0000, A 0.000, B 0.000, C 0.000 }
gfCNCPoint2[12484] = {X 337.4845, Y 30.0811, Z -3.0000, A 0.000, B 0.000, C 0.000 }
gfCNCPoint2[12485] = {X 338.1274, Y 30.8804, Z -3.0000, A 0.000, B 0.000, C 0.000 }
gfCNCPoint2[12486] = {X 338.5677, Y 31.8067, Z -3.0000, A 0.000, B 0.000, C 0.000 }
gfCNCPoint2[12487] = {X 338.7817, Y 32.8099, Z -3.0000, A 0.000, B 0.000, C 0.000 }
gfCNCPoint2[12488] = {X 338.7575, Y 33.8353, Z -3.0000, A 0.000, B 0.000, C 0.000 }
gfCNCPoint2[12489] = {X 339.5034, Y 34.5089, Z -3.0000, A 0.000, B 0.000, C 0.000 }
gfCNCPoint2[12490] = {X 340.2819, Y 35.1446, Z -3.0000, A 0.000, B 0.000, C 0.000 }
gfCNCPoint2[12491] = {X 341.4932, Y 35.9469, Z -3.0000, A 0.000, B 0.000, C 0.000 }
gfCNCPoint2[12492] = {X 342.8033, Y 36.5750, Z -3.0000, A 0.000, B 0.000, C 0.000 }
gfCNCPoint2[12493] = {X 344.1875, Y 37.0168, Z -3.0000, A 0.000, B 0.000, C 0.000 }
gfCNCPoint2[12494] = {X 345.6192, Y 37.2639, Z -3.0000, A 0.000, B 0.000, C 0.000 }
gfCNCPoint2[12495] = {X 347.0713, Y 37.3118, Z -3.0000, A 0.000, B 0.000, C 0.000 }
gfCNCPoint2[12496] = {X 347.5137, Y 37.2889, Z -3.0000, A 0.000, B 0.000, C 0.000 }
gfCNCPoint2[12497] = {X 348.9406, Y 37.0973, Z -3.0000, A 0.000, B 0.000, C 0.000 }
gfCNCPoint2[12498] = {X 350.3174, Y 36.6761, Z -3.0000, A 0.000, B 0.000, C 0.000 }
gfCNCPoint2[12499] = {X 351.6072, Y 36.0363, Z -3.0000, A 0.000, B 0.000, C 0.000 }
gfCNCPoint2[12500] = {X 352.7757, Y 35.1952, Z -3.0000, A 0.000, B 0.000, C 0.000 }
gfCNCPoint2[12501] = {X 353.9224, Y 34.0816, Z -3.0000, A 0.000, B 0.000, C 0.000 }
gfCNCPoint2[12502] = {X 354.9147, Y 32.8285, Z -3.0000, A 0.000, B 0.000, C 0.000 }
gfCNCPoint2[12503] = {X 355.7359, Y 31.4572, Z -3.0000, A 0.000, B 0.000, C 0.000 }
gfCNCPoint2[12504] = {X 356.3721, Y 29.9909, Z -3.0000, A 0.000, B 0.000, C 0.000 }
gfCNCPoint2[12505] = {X 356.8126, Y 28.4543, Z -3.0000, A 0.000, B 0.000, C 0.000 }
gfCNCPoint2[12506] = {X 357.0847, Y 26.7730, Z -3.0000, A 0.000, B 0.000, C 0.000 }
gfCNCPoint2[12507] = {X 357.1955, Y 25.0733, Z -3.0000, A 0.000, B 0.000, C 0.000 }
gfCNCPoint2[12508] = {X 357.1438, Y 23.3709, Z -3.0000, A 0.000, B 0.000, C 0.000 }
gfCNCPoint2[12509] = {X 356.9303, Y 21.6811, Z -3.0000, A 0.000, B 0.000, C 0.000 }
gfCNCPoint2[12510] = {X 356.5961, Y 20.2415, Z -3.0000, A 0.000, B 0.000, C 0.000 }
gfCNCPoint2[12511] = {X 356.0863, Y 18.8543, Z -3.0000, A 0.000, B 0.000, C 0.000 }
gfCNCPoint2[12512] = {X 355.4089, Y 17.5409, Z -3.0000, A 0.000, B 0.000, C 0.000 }
gfCNCPoint2[12513] = {X 354.5740, Y 16.3214, Z -3.0000, A 0.000, B 0.000, C 0.000 }
gfCNCPoint2[12514] = {X 353.6959, Y 15.3422, Z -3.0000, A 0.000, B 0.000, C 0.000 }
gfCNCPoint2[12515] = {X 352.6865, Y 14.4988, Z -3.0000, A 0.000, B 0.000, C 0.000 }
gfCNCPoint2[12516] = {X 351.5667, Y 13.8087, Z -3.0000, A 0.000, B 0.000, C 0.000 }
gfCNCPoint2[12517] = {X 350.3596, Y 13.2862, Z -3.0000, A 0.000, B 0.000, C 0.000 }
gfCNCPoint2[12518] = {X 349.0902, Y 12.9419, Z -3.0000, A 0.000, B 0.000, C 0.000 }
gfCNCPoint2[12519] = {X 347.3475, Y 12.7247, Z -3.0000, A 0.000, B 0.000, C 0.000 }
gfCNCPoint2[12520] = {X 345.5915, Y 12.7391, Z -3.0000, A 0.000, B 0.000, C 0.000 }
gfCNCPoint2[12521] = {X 343.8526, Y 12.9845, Z -3.0000, A 0.000, B 0.000, C 0.000 }
gfCNCPoint2[12522] = {X 342.1613, Y 13.4569, Z -3.0000, A 0.000, B 0.000, C 0.000 }
gfCNCPoint2[12523] = {X 340.5469, Y 14.1480, Z -3.0000, A 0.000, B 0.000, C 0.000 }
gfCNCPoint2[12524] = {X 339.0375, Y 15.0457, Z -3.0000, A 0.000, B 0.000, C 0.000 }
gfCNCPoint2[12525] = {X 338.9897, Y 15.9038, Z -3.0000, A 0.000, B 0.000, C 0.000 }
gfCNCPoint2[12526] = {X 338.7759, Y 16.7362, Z -3.0000, A 0.000, B 0.000, C 0.000 }
gfCNCPoint2[12527] = {X 338.4044, Y 17.5111, Z -3.0000, A 0.000, B 0.000, C 0.000 }
gfCNCPoint2[12528] = {X 337.8894, Y 18.1991, Z -3.0000, A 0.000, B 0.000, C 0.000 }
gfCNCPoint2[12529] = {X 337.2504, Y 18.7738, Z -3.0000, A 0.000, B 0.000, C 0.000 }
gfCNCPoint2[12530] = {X 336.5606, Y 19.2813, Z -3.0000, A 0.000, B 0.000, C 0.000 }
gfCNCPoint2[12531] = {X 335.7284, Y 19.7495, Z -3.0000, A 0.000, B 0.000, C 0.000 }
gfCNCPoint2[12532] = {X 334.8148, Y 20.0271, Z -3.0000, A 0.000, B 0.000, C 0.000 }
gfCNCPoint2[12533] = {X 333.8628, Y 20.1012, Z -3.0000, A 0.000, B 0.000, C 0.000 }
gfCNCPoint2[12534] = {X 332.9173, Y 19.9681, Z -3.0000, A 0.000, B 0.000, C 0.000 }
gfCNCPoint2[12535] = {X 332.0228, Y 19.6341, Z -3.0000, A 0.000, B 0.000, C 0.000 }
gfCNCPoint2[12536] = {X 331.2213, Y 19.1151, Z -3.0000, A 0.000, B 0.000, C 0.000 }
gfCNCPoint2[12537] = {X 330.5507, Y 18.4353, Z -3.0000, A 0.000, B 0.000, C 0.000 }
gfCNCPoint2[12538] = {X 330.0425, Y 17.6269, Z -3.0000, A 0.000, B 0.000, C 0.000 }
gfCNCPoint2[12539] = {X 326.5223, Y 10.3852, Z -3.0000, A 0.000, B 0.000, C 0.000 }
gfCNCPoint2[12540] = {X 326.2154, Y 9.5469, Z -3.0000, A 0.000, B 0.000, C 0.000 }
gfCNCPoint2[12541] = {X 326.0841, Y 8.6639, Z -3.0000, A 0.000, B 0.000, C 0.000 }
gfCNCPoint2[12542] = {X 326.1338, Y 7.7725, Z -3.0000, A 0.000, B 0.000, C 0.000 }
gfCNCPoint2[12543] = {X 326.3623, Y 6.9096, Z -3.0000, A 0.000, B 0.000, C 0.000 }
gfCNCPoint2[12544] = {X 326.7603, Y 6.1105, Z -3.0000, A 0.000, B 0.000, C 0.000 }
gfCNCPoint2[12545] = {X 327.3114, Y 5.4082, Z -3.0000, A 0.000, B 0.000, C 0.000 }
gfCNCPoint2[12546] = {X 327.9929, Y 4.8316, Z -3.0000, A 0.000, B 0.000, C 0.000 }
gfCNCPoint2[12547] = {X 328.6647, Y 4.3715, Z -3.0000, A 0.000, B 0.000, C 0.000 }
gfCNCPoint2[12548] = {X 329.5526, Y 3.9111, Z -3.0000, A 0.000, B 0.000, C 0.000 }
gfCNCPoint2[12549] = {X 330.5215, Y 3.6630, Z -3.0000, A 0.000, B 0.000, C 0.000 }
gfCNCPoint2[12550] = {X 331.5214, Y 3.6402, Z -3.0000, A 0.000, B 0.000, C 0.000 }
gfCNCPoint2[12551] = {X 332.5006, Y 3.8438, Z -3.0000, A 0.000, B 0.000, C 0.000 }
gfCNCPoint2[12552] = {X 333.5108, Y 3.2690, Z -3.0000, A 0.000, B 0.000, C 0.000 }
gfCNCPoint2[12553] = {X 334.5436, Y 2.7360, Z -3.0000, A 0.000, B 0.000, C 0.000 }
gfCNCPoint2[12554] = {X 334.3322, Y 2.3050, Z -3.0000, A 0.000, B 0.000, C 0.000 }
gfCNCPoint2[12555] = {X 2.3035, Y 2.3050, Z -3.0000, A 0.000, B 0.000, C 0.000 }
gfCNCPoint2[12556] = {X 2.3035, Y 6.8597, Z -3.0000, A 0.000, B 0.000, C 0.000 }
gfCNCPoint2[12557] = {X 2.4106, Y 6.8811, Z -3.0000, A 0.000, B 0.000, C 0.000 }
gfCNCPoint2[12558] = {X 2.8637, Y 6.6950, Z -3.0000, A 0.000, B 0.000, C 0.000 }
gfCNCPoint2[12559] = {X 3.3223, Y 6.5230, Z -3.0000, A 0.000, B 0.000, C 0.000 }
gfCNCPoint2[12560] = {X 5.4290, Y 5.7897, Z -3.0000, A 0.000, B 0.000, C 0.000 }
gfCNCPoint2[12561] = {X 7.5909, Y 5.2402, Z -3.0000, A 0.000, B 0.000, C 0.000 }
gfCNCPoint2[12562] = {X 9.7920, Y 4.8785, Z -3.0000, A 0.000, B 0.000, C 0.000 }
gfCNCPoint2[12563] = {X 12.0161, Y 4.7072, Z -3.0000, A 0.000, B 0.000, C 0.000 }
gfCNCPoint2[12564] = {X 14.2466, Y 4.7278, Z -3.0000, A 0.000, B 0.000, C 0.000 }
gfCNCPoint2[12565] = {X 16.4671, Y 4.9399, Z -3.0000, A 0.000, B 0.000, C 0.000 }
gfCNCPoint2[12566] = {X 18.0961, Y 5.2207, Z -3.0000, A 0.000, B 0.000, C 0.000 }
gfCNCPoint2[12567] = {X 19.6962, Y 5.6354, Z -3.0000, A 0.000, B 0.000, C 0.000 }
gfCNCPoint2[12568] = {X 21.2565, Y 6.1813, Z -3.0000, A 0.000, B 0.000, C 0.000 }
gfCNCPoint2[12569] = {X 22.7661, Y 6.8545, Z -3.0000, A 0.000, B 0.000, C 0.000 }
gfCNCPoint2[12570] = {X 24.4880, Y 7.8187, Z -3.0000, A 0.000, B 0.000, C 0.000 }
gfCNCPoint2[12571] = {X 26.1061, Y 8.9485, Z -3.0000, A 0.000, B 0.000, C 0.000 }
gfCNCPoint2[12572] = {X 27.4002, Y 10.0786, Z -3.0000, A 0.000, B 0.000, C 0.000 }
gfCNCPoint2[12573] = {X 28.5611, Y 11.3452, Z -3.0000, A 0.000, B 0.000, C 0.000 }
gfCNCPoint2[12574] = {X 29.5744, Y 12.7327, Z -3.0000, A 0.000, B 0.000, C 0.000 }
gfCNCPoint2[12575] = {X 30.4276, Y 14.2240, Z -3.0000, A 0.000, B 0.000, C 0.000 }
gfCNCPoint2[12576] = {X 31.1101, Y 15.8007, Z -3.0000, A 0.000, B 0.000, C 0.000 }
gfCNCPoint2[12577] = {X 31.6695, Y 17.7363, Z -3.0000, A 0.000, B 0.000, C 0.000 }
gfCNCPoint2[12578] = {X 32.0025, Y 19.7233, Z -3.0000, A 0.000, B 0.000, C 0.000 }
gfCNCPoint2[12579] = {X 32.1048, Y 21.7354, Z -3.0000, A 0.000, B 0.000, C 0.000 }
gfCNCPoint2[12580] = {X 31.9751, Y 23.7460, Z -3.0000, A 0.000, B 0.000, C 0.000 }
gfCNCPoint2[12581] = {X 31.6149, Y 25.7283, Z -3.0000, A 0.000, B 0.000, C 0.000 }
gfCNCPoint2[12582] = {X 31.1961, Y 27.1573, Z -3.0000, A 0.000, B 0.000, C 0.000 }
gfCNCPoint2[12583] = {X 30.6297, Y 28.5345, Z -3.0000, A 0.000, B 0.000, C 0.000 }
gfCNCPoint2[12584] = {X 29.9219, Y 29.8446, Z -3.0000, A 0.000, B 0.000, C 0.000 }
gfCNCPoint2[12585] = {X 29.0805, Y 31.0732, Z -3.0000, A 0.000, B 0.000, C 0.000 }
gfCNCPoint2[12586] = {X 29.6383, Y 31.7916, Z -3.0000, A 0.000, B 0.000, C 0.000 }
gfCNCPoint2[12587] = {X 30.0953, Y 32.5781, Z -3.0000, A 0.000, B 0.000, C 0.000 }
gfCNCPoint2[12588] = {X 33.1423, Y 38.8726, Z -3.0000, A 0.000, B 0.000, C 0.000 }
gfCNCPoint2[12589] = {X 33.5391, Y 39.8957, Z -3.0000, A 0.000, B 0.000, C 0.000 }
gfCNCPoint2[12590] = {X 33.7662, Y 40.9694, Z -3.0000, A 0.000, B 0.000, C 0.000 }
gfCNCPoint2[12591] = {X 33.8177, Y 42.0656, Z -3.0000, A 0.000, B 0.000, C 0.000 }
gfCNCPoint2[12592] = {X 33.7164, Y 43.0266, Z -3.0000, A 0.000, B 0.000, C 0.000 }
gfCNCPoint2[12593] = {X 33.4799, Y 43.9636, Z -3.0000, A 0.000, B 0.000, C 0.000 }
gfCNCPoint2[12594] = {X 33.1103, Y 44.8630, Z -3.0000, A 0.000, B 0.000, C 0.000 }
gfCNCPoint2[12595] = {X 32.6161, Y 45.7005, Z -3.0000, A 0.000, B 0.000, C 0.000 }
gfCNCPoint2[12596] = {X 32.0075, Y 46.4590, Z -3.0000, A 0.000, B 0.000, C 0.000 }
gfCNCPoint2[12597] = {X 31.2970, Y 47.1229, Z -3.0000, A 0.000, B 0.000, C 0.000 }
gfCNCPoint2[12598] = {X 30.7587, Y 47.5582, Z -3.0000, A 0.000, B 0.000, C 0.000 }
gfCNCPoint2[12599] = {X 29.8532, Y 48.1756, Z -3.0000, A 0.000, B 0.000, C 0.000 }
gfCNCPoint2[12600] = {X 28.8604, Y 48.6399, Z -3.0000, A 0.000, B 0.000, C 0.000 }
gfCNCPoint2[12601] = {X 27.8060, Y 48.9391, Z -3.0000, A 0.000, B 0.000, C 0.000 }
gfCNCPoint2[12602] = {X 26.7173, Y 49.0654, Z -3.0000, A 0.000, B 0.000, C 0.000 }
gfCNCPoint2[12603] = {X 25.6225, Y 49.0157, Z -3.0000, A 0.000, B 0.000, C 0.000 }
gfCNCPoint2[12604] = {X 23.4251, Y 50.0829, Z -3.0000, A 0.000, B 0.000, C 0.000 }
gfCNCPoint2[12605] = {X 21.1492, Y 50.9706, Z -3.0000, A 0.000, B 0.000, C 0.000 }
gfCNCPoint2[12606] = {X 19.0233, Y 51.6404, Z -3.0000, A 0.000, B 0.000, C 0.000 }
gfCNCPoint2[12607] = {X 16.8467, Y 52.1204, Z -3.0000, A 0.000, B 0.000, C 0.000 }
gfCNCPoint2[12608] = {X 14.6363, Y 52.4070, Z -3.0000, A 0.000, B 0.000, C 0.000 }
gfCNCPoint2[12609] = {X 12.4093, Y 52.4979, Z -3.0000, A 0.000, B 0.000, C 0.000 }
gfCNCPoint2[12610] = {X 10.1829, Y 52.3925, Z -3.0000, A 0.000, B 0.000, C 0.000 }
gfCNCPoint2[12611] = {X 7.9745, Y 52.0915, Z -3.0000, A 0.000, B 0.000, C 0.000 }
gfCNCPoint2[12612] = {X 6.6902, Y 51.8235, Z -3.0000, A 0.000, B 0.000, C 0.000 }
gfCNCPoint2[12613] = {X 5.4266, Y 51.4702, Z -3.0000, A 0.000, B 0.000, C 0.000 }
gfCNCPoint2[12614] = {X 3.8372, Y 50.8914, Z -3.0000, A 0.000, B 0.000, C 0.000 }
gfCNCPoint2[12615] = {X 2.3035, Y 50.1779, Z -3.0000, A 0.000, B 0.000, C 0.000 }
gfCNCPoint2[12616] = {X 2.3035, Y 97.6950, Z -3.0000, A 0.000, B 0.000, C 0.000 }
gfCNCPoint2[12617] = {X 120.1200, Y 97.6950, Z -3.0000, A 0.000, B 0.000, C 0.000 }
gfCNCPoint2[12618] = {X 120.1200, Y 97.0659, Z -3.0000, A 0.000, B 0.000, C 0.000 }
gfCNCPoint2[12619] = {X 120.2339, Y 96.0177, Z -3.0000, A 0.000, B 0.000, C 0.000 }
gfCNCPoint2[12620] = {X 120.5703, Y 95.0184, Z -3.0000, A 0.000, B 0.000, C 0.000 }
gfCNCPoint2[12621] = {X 121.1136, Y 94.1146, Z -3.0000, A 0.000, B 0.000, C 0.000 }
gfCNCPoint2[12622] = {X 121.8383, Y 93.3487, Z -3.0000, A 0.000, B 0.000, C 0.000 }
gfCNCPoint2[12623] = {X 122.7105, Y 92.7563, Z -3.0000, A 0.000, B 0.000, C 0.000 }
gfCNCPoint2[12624] = {X 123.6897, Y 92.3651, Z -3.0000, A 0.000, B 0.000, C 0.000 }
gfCNCPoint2[12625] = {X 124.7301, Y 92.1934, Z -3.0000, A 0.000, B 0.000, C 0.000 }
gfCNCPoint2[12626] = {X 124.7875, Y 92.1788, Z -3.0000, A 0.000, B 0.000, C 0.000 }
gfCNCPoint2[12627] = {X 124.8458, Y 92.1682, Z -3.0000, A 0.000, B 0.000, C 0.000 }
gfCNCPoint2[12628] = {X 125.3649, Y 92.0912, Z -3.0000, A 0.000, B 0.000, C 0.000 }
gfCNCPoint2[12629] = {X 126.1000, Y 91.9694, Z -3.0000, A 0.000, B 0.000, C 0.000 }
gfCNCPoint2[12630] = {X 126.8261, Y 91.8022, Z -3.0000, A 0.000, B 0.000, C 0.000 }
gfCNCPoint2[12631] = {X 127.9740, Y 90.7129, Z -3.0000, A 0.000, B 0.000, C 0.000 }
gfCNCPoint2[12632] = {X 129.0636, Y 89.5653, Z -3.0000, A 0.000, B 0.000, C 0.000 }
gfCNCPoint2[12633] = {X 154.9463, Y 61.1425, Z -3.0000, A 0.000, B 0.000, C 0.000 }
gfCNCPoint2[12634] = {X 154.6593, Y 60.4498, Z -3.0000, A 0.000, B 0.000, C 0.000 }
gfCNCPoint2[12635] = {X 154.4819, Y 59.7214, Z -3.0000, A 0.000, B 0.000, C 0.000 }
gfCNCPoint2[12636] = {X 154.4181, Y 58.9744, Z -3.0000, A 0.000, B 0.000, C 0.000 }
gfCNCPoint2[12637] = {X 154.4180, Y 58.0000, Z -3.0000, A 0.000, B 0.000, C 0.000 }
gfCNCPoint2[12638] = {X 154.5117, Y 57.0480, Z -3.0000, A 0.000, B 0.000, C 0.000 }
gfCNCPoint2[12639] = {X 154.7894, Y 56.1325, Z -3.0000, A 0.000, B 0.000, C 0.000 }
gfCNCPoint2[12640] = {X 155.2404, Y 55.2888, Z -3.0000, A 0.000, B 0.000, C 0.000 }
gfCNCPoint2[12641] = {X 155.8473, Y 54.5493, Z -3.0000, A 0.000, B 0.000, C 0.000 }
gfCNCPoint2[12642] = {X 156.5868, Y 53.9424, Z -3.0000, A 0.000, B 0.000, C 0.000 }
gfCNCPoint2[12643] = {X 157.4305, Y 53.4915, Z -3.0000, A 0.000, B 0.000, C 0.000 }
gfCNCPoint2[12644] = {X 158.3459, Y 53.2138, Z -3.0000, A 0.000, B 0.000, C 0.000 }
gfCNCPoint2[12645] = {X 159.2980, Y 53.1200, Z -3.0000, A 0.000, B 0.000, C 0.000 }
gfCNCPoint2[12646] = {X 178.5335, Y 53.1200, Z -3.0000, A 0.000, B 0.000, C 0.000 }
gfCNCPoint2[12647] = {X 179.4855, Y 53.2138, Z -3.0000, A 0.000, B 0.000, C 0.000 }
gfCNCPoint2[12648] = {X 180.4010, Y 53.4915, Z -3.0000, A 0.000, B 0.000, C 0.000 }
gfCNCPoint2[12649] = {X 181.2447, Y 53.9424, Z -3.0000, A 0.000, B 0.000, C 0.000 }
gfCNCPoint2[12650] = {X 181.9842, Y 54.5493, Z -3.0000, A 0.000, B 0.000, C 0.000 }
gfCNCPoint2[12651] = {X 182.5911, Y 55.2888, Z -3.0000, A 0.000, B 0.000, C 0.000 }
gfCNCPoint2[12652] = {X 183.0420, Y 56.1325, Z -3.0000, A 0.000, B 0.000, C 0.000 }
gfCNCPoint2[12653] = {X 183.3197, Y 57.0480, Z -3.0000, A 0.000, B 0.000, C 0.000 }
gfCNCPoint2[12654] = {X 183.4135, Y 58.0000, Z -3.0000, A 0.000, B 0.000, C 0.000 }
gfCNCPoint2[12655] = {X 183.4133, Y 58.9744, Z -3.0000, A 0.000, B 0.000, C 0.000 }
gfCNCPoint2[12656] = {X 183.3512, Y 59.7114, Z -3.0000, A 0.000, B 0.000, C 0.000 }
gfCNCPoint2[12657] = {X 183.1784, Y 60.4306, Z -3.0000, A 0.000, B 0.000, C 0.000 }
gfCNCPoint2[12658] = {X 182.8988, Y 61.1154, Z -3.0000, A 0.000, B 0.000, C 0.000 }
gfCNCPoint2[12659] = {X 209.8909, Y 90.5757, Z -3.0000, A 0.000, B 0.000, C 0.000 }
gfCNCPoint2[12660] = {X 210.5200, Y 91.2140, Z -3.0000, A 0.000, B 0.000, C 0.000 }
gfCNCPoint2[12661] = {X 211.1939, Y 91.8048, Z -3.0000, A 0.000, B 0.000, C 0.000 }
gfCNCPoint2[12662] = {X 211.3598, Y 91.9090, Z -3.0000, A 0.000, B 0.000, C 0.000 }
gfCNCPoint2[12663] = {X 211.5461, Y 91.9699, Z -3.0000, A 0.000, B 0.000, C 0.000 }
gfCNCPoint2[12664] = {X 212.2018, Y 92.1101, Z -3.0000, A 0.000, B 0.000, C 0.000 }
gfCNCPoint2[12665] = {X 213.4083, Y 92.2621, Z -3.0000, A 0.000, B 0.000, C 0.000 }
gfCNCPoint2[12666] = {X 214.4424, Y 92.1759, Z -3.0000, A 0.000, B 0.000, C 0.000 }
gfCNCPoint2[12667] = {X 215.4785, Y 92.1170, Z -3.0000, A 0.000, B 0.000, C 0.000 }
gfCNCPoint2[12668] = {X 216.0525, Y 92.0571, Z -3.0000, A 0.000, B 0.000, C 0.000 }
gfCNCPoint2[12669] = {X 216.6054, Y 91.8918, Z -3.0000, A 0.000, B 0.000, C 0.000 }
gfCNCPoint2[12670] = {X 217.1180, Y 91.6268, Z -3.0000, A 0.000, B 0.000, C 0.000 }
gfCNCPoint2[12671] = {X 244.6016, Y 74.0195, Z -3.0000, A 0.000, B 0.000, C 0.000 }
gfCNCPoint2[12672] = {X 221.4278, Y 64.9251, Z -3.0000, A 0.000, B 0.000, C 0.000 }
gfCNCPoint2[12673] = {X 219.7200, Y 64.3529, Z -3.0000, A 0.000, B 0.000, C 0.000 }
gfCNCPoint2[12674] = {X 217.9579, Y 63.9800, Z -3.0000, A 0.000, B 0.000, C 0.000 }
gfCNCPoint2[12675] = {X 216.1647, Y 63.8112, Z -3.0000, A 0.000, B 0.000, C 0.000 }
gfCNCPoint2[12676] = {X 215.1121, Y 63.6594, Z -3.0000, A 0.000, B 0.000, C 0.000 }
gfCNCPoint2[12677] = {X 214.1174, Y 63.2832, Z -3.0000, A 0.000, B 0.000, C 0.000 }
gfCNCPoint2[12678] = {X 213.2278, Y 62.7005, Z -3.0000, A 0.000, B 0.000, C 0.000 }
gfCNCPoint2[12679] = {X 212.4856, Y 61.9389, Z -3.0000, A 0.000, B 0.000, C 0.000 }
gfCNCPoint2[12680] = {X 211.9260, Y 61.0346, Z -3.0000, A 0.000, B 0.000, C 0.000 }
gfCNCPoint2[12681] = {X 211.5756, Y 60.0305, Z -3.0000, A 0.000, B 0.000, C 0.000 }
gfCNCPoint2[12682] = {X 211.4510, Y 58.9744, Z -3.0000, A 0.000, B 0.000, C 0.000 }
gfCNCPoint2[12683] = {X 211.4508, Y 58.0000, Z -3.0000, A 0.000, B 0.000, C 0.000 }
gfCNCPoint2[12684] = {X 211.5446, Y 57.0480, Z -3.0000, A 0.000, B 0.000, C 0.000 }
gfCNCPoint2[12685] = {X 211.8223, Y 56.1325, Z -3.0000, A 0.000, B 0.000, C 0.000 }
gfCNCPoint2[12686] = {X 212.2732, Y 55.2888, Z -3.0000, A 0.000, B 0.000, C 0.000 }
gfCNCPoint2[12687] = {X 212.8801, Y 54.5493, Z -3.0000, A 0.000, B 0.000, C 0.000 }
gfCNCPoint2[12688] = {X 213.6196, Y 53.9424, Z -3.0000, A 0.000, B 0.000, C 0.000 }
gfCNCPoint2[12689] = {X 214.4633, Y 53.4915, Z -3.0000, A 0.000, B 0.000, C 0.000 }
gfCNCPoint2[12690] = {X 215.3788, Y 53.2138, Z -3.0000, A 0.000, B 0.000, C 0.000 }
gfCNCPoint2[12691] = {X 216.3308, Y 53.1200, Z -3.0000, A 0.000, B 0.000, C 0.000 }
gfCNCPoint2[12692] = {X 237.2617, Y 53.1200, Z -3.0000, A 0.000, B 0.000, C 0.000 }
gfCNCPoint2[12693] = {X 238.3265, Y 53.2376, Z -3.0000, A 0.000, B 0.000, C 0.000 }
gfCNCPoint2[12694] = {X 239.3401, Y 53.5847, Z -3.0000, A 0.000, B 0.000, C 0.000 }
gfCNCPoint2[12695] = {X 240.2535, Y 54.1446, Z -3.0000, A 0.000, B 0.000, C 0.000 }
gfCNCPoint2[12696] = {X 241.0226, Y 54.8904, Z -3.0000, A 0.000, B 0.000, C 0.000 }
gfCNCPoint2[12697] = {X 241.6105, Y 55.7860, Z -3.0000, A 0.000, B 0.000, C 0.000 }
gfCNCPoint2[12698] = {X 241.9889, Y 56.7883, Z -3.0000, A 0.000, B 0.000, C 0.000 }
gfCNCPoint2[12699] = {X 242.1394, Y 57.8490, Z -3.0000, A 0.000, B 0.000, C 0.000 }
gfCNCPoint2[12700] = {X 247.6957, Y 60.0151, Z -3.0000, A 0.000, B 0.000, C 0.000 }
gfCNCPoint2[12701] = {X 275.0734, Y 70.8780, Z -3.0000, A 0.000, B 0.000, C 0.000 }
gfCNCPoint2[12702] = {X 275.0728, Y 63.6742, Z -3.0000, A 0.000, B 0.000, C 0.000 }
gfCNCPoint2[12703] = {X 274.0645, Y 63.3059, Z -3.0000, A 0.000, B 0.000, C 0.000 }
gfCNCPoint2[12704] = {X 273.1610, Y 62.7261, Z -3.0000, A 0.000, B 0.000, C 0.000 }
gfCNCPoint2[12705] = {X 272.4062, Y 61.9627, Z -3.0000, A 0.000, B 0.000, C 0.000 }
gfCNCPoint2[12706] = {X 271.8366, Y 61.0528, Z -3.0000, A 0.000, B 0.000, C 0.000 }
gfCNCPoint2[12707] = {X 271.4797, Y 60.0404, Z -3.0000, A 0.000, B 0.000, C 0.000 }
gfCNCPoint2[12708] = {X 271.3529, Y 58.9744, Z -3.0000, A 0.000, B 0.000, C 0.000 }
gfCNCPoint2[12709] = {X 271.3527, Y 58.0000, Z -3.0000, A 0.000, B 0.000, C 0.000 }
gfCNCPoint2[12710] = {X 271.4465, Y 57.0480, Z -3.0000, A 0.000, B 0.000, C 0.000 }
gfCNCPoint2[12711] = {X 271.7242, Y 56.1325, Z -3.0000, A 0.000, B 0.000, C 0.000 }
gfCNCPoint2[12712] = {X 272.1751, Y 55.2888, Z -3.0000, A 0.000, B 0.000, C 0.000 }
gfCNCPoint2[12713] = {X 272.7820, Y 54.5493, Z -3.0000, A 0.000, B 0.000, C 0.000 }
gfCNCPoint2[12714] = {X 273.5215, Y 53.9424, Z -3.0000, A 0.000, B 0.000, C 0.000 }
gfCNCPoint2[12715] = {X 274.3652, Y 53.4915, Z -3.0000, A 0.000, B 0.000, C 0.000 }
gfCNCPoint2[12716] = {X 275.2806, Y 53.2138, Z -3.0000, A 0.000, B 0.000, C 0.000 }
gfCNCPoint2[12717] = {X 276.2327, Y 53.1200, Z -3.0000, A 0.000, B 0.000, C 0.000 }
gfCNCPoint2[12718] = {X 292.7731, Y 53.1200, Z -3.0000, A 0.000, B 0.000, C 0.000 }
gfCNCPoint2[12719] = {X 293.7251, Y 53.2138, Z -3.0000, A 0.000, B 0.000, C 0.000 }
gfCNCPoint2[12720] = {X 294.6406, Y 53.4915, Z -3.0000, A 0.000, B 0.000, C 0.000 }
gfCNCPoint2[12721] = {X 295.4843, Y 53.9424, Z -3.0000, A 0.000, B 0.000, C 0.000 }
gfCNCPoint2[12722] = {X 296.2238, Y 54.5493, Z -3.0000, A 0.000, B 0.000, C 0.000 }
gfCNCPoint2[12723] = {X 296.8307, Y 55.2888, Z -3.0000, A 0.000, B 0.000, C 0.000 }
gfCNCPoint2[12724] = {X 297.2816, Y 56.1325, Z -3.0000, A 0.000, B 0.000, C 0.000 }
gfCNCPoint2[12725] = {X 297.5593, Y 57.0480, Z -3.0000, A 0.000, B 0.000, C 0.000 }
gfCNCPoint2[12726] = {X 297.6531, Y 58.0000, Z -3.0000, A 0.000, B 0.000, C 0.000 }
gfCNCPoint2[12727] = {X 297.6531, Y 58.9371, Z -3.0000, A 0.000, B 0.000, C 0.000 }
gfCNCPoint2[12728] = {X 297.5306, Y 60.0092, Z -3.0000, A 0.000, B 0.000, C 0.000 }
gfCNCPoint2[12729] = {X 297.1762, Y 61.0285, Z -3.0000, A 0.000, B 0.000, C 0.000 }
gfCNCPoint2[12730] = {X 296.6072, Y 61.9455, Z -3.0000, A 0.000, B 0.000, C 0.000 }
gfCNCPoint2[12731] = {X 295.8511, Y 62.7155, Z -3.0000, A 0.000, B 0.000, C 0.000 }
gfCNCPoint2[12732] = {X 294.9447, Y 63.3012, Z -3.0000, A 0.000, B 0.000, C 0.000 }
gfCNCPoint2[12733] = {X 293.9321, Y 63.6742, Z -3.0000, A 0.000, B 0.000, C 0.000 }
gfCNCPoint2[12734] = {X 293.9321, Y 92.3206, Z -3.0000, A 0.000, B 0.000, C 0.000 }
gfCNCPoint2[12735] = {X 294.9446, Y 92.6962, Z -3.0000, A 0.000, B 0.000, C 0.000 }
gfCNCPoint2[12736] = {X 295.8506, Y 93.2839, Z -3.0000, A 0.000, B 0.000, C 0.000 }
gfCNCPoint2[12737] = {X 296.6063, Y 94.0553, Z -3.0000, A 0.000, B 0.000, C 0.000 }
gfCNCPoint2[12738] = {X 297.1752, Y 94.9732, Z -3.0000, A 0.000, B 0.000, C 0.000 }
gfCNCPoint2[12739] = {X 297.5299, Y 95.9932, Z -3.0000, A 0.000, B 0.000, C 0.000 }
gfCNCPoint2[12740] = {X 297.6531, Y 97.0661, Z -3.0000, A 0.000, B 0.000, C 0.000 }
gfCNCPoint2[12741] = {X 297.6531, Y 97.6950, Z -3.0000, A 0.000, B 0.000, C 0.000 }
gfCNCPoint2[12742] = {X 297.1731, Y 97.6950, Z -3.0000, A 0.000, B 0.000, C 0.000 }
gfCNCPoint2[12743] = {X 297.1731, Y 98.0000, Z -3.0000, A 0.000, B 0.000, C 0.000 }
gfCNCPoint2[12744] = {X 297.0628, Y 98.9791, Z -3.0000, A 0.000, B 0.000, C 0.000 }
gfCNCPoint2[12745] = {X 296.7373, Y 99.9091, Z -3.0000, A 0.000, B 0.000, C 0.000 }
gfCNCPoint2[12746] = {X 296.2131, Y 100.7434, Z -3.0000, A 0.000, B 0.000, C 0.000 }
gfCNCPoint2[12747] = {X 295.5164, Y 101.4401, Z -3.0000, A 0.000, B 0.000, C 0.000 }
gfCNCPoint2[12748] = {X 294.6822, Y 101.9643, Z -3.0000, A 0.000, B 0.000, C 0.000 }
gfCNCPoint2[12749] = {X 293.7522, Y 102.2897, Z -3.0000, A 0.000, B 0.000, C 0.000 }
gfCNCPoint2[12750] = {X 292.7731, Y 102.4000, Z -3.0000, A 0.000, B 0.000, C 0.000 }
gfCNCPoint2[12751] = {X 276.2327, Y 102.4000, Z -3.0000, A 0.000, B 0.000, C 0.000 }
gfCNCPoint2[12752] = {X 275.2536, Y 102.2897, Z -3.0000, A 0.000, B 0.000, C 0.000 }
gfCNCPoint2[12753] = {X 274.3236, Y 101.9643, Z -3.0000, A 0.000, B 0.000, C 0.000 }
gfCNCPoint2[12754] = {X 273.4893, Y 101.4401, Z -3.0000, A 0.000, B 0.000, C 0.000 }
gfCNCPoint2[12755] = {X 272.7926, Y 100.7434, Z -3.0000, A 0.000, B 0.000, C 0.000 }
gfCNCPoint2[12756] = {X 272.2684, Y 99.9091, Z -3.0000, A 0.000, B 0.000, C 0.000 }
gfCNCPoint2[12757] = {X 271.9430, Y 98.9791, Z -3.0000, A 0.000, B 0.000, C 0.000 }
gfCNCPoint2[12758] = {X 271.8327, Y 98.0000, Z -3.0000, A 0.000, B 0.000, C 0.000 }
gfCNCPoint2[12759] = {X 271.8329, Y 97.0190, Z -3.0000, A 0.000, B 0.000, C 0.000 }
gfCNCPoint2[12760] = {X 271.9305, Y 96.1432, Z -3.0000, A 0.000, B 0.000, C 0.000 }
gfCNCPoint2[12761] = {X 272.2006, Y 95.3045, Z -3.0000, A 0.000, B 0.000, C 0.000 }
gfCNCPoint2[12762] = {X 272.6325, Y 94.5364, Z -3.0000, A 0.000, B 0.000, C 0.000 }
gfCNCPoint2[12763] = {X 273.2087, Y 93.8698, Z -3.0000, A 0.000, B 0.000, C 0.000 }
gfCNCPoint2[12764] = {X 273.9062, Y 93.3313, Z -3.0000, A 0.000, B 0.000, C 0.000 }
gfCNCPoint2[12765] = {X 274.6970, Y 92.9426, Z -3.0000, A 0.000, B 0.000, C 0.000 }
gfCNCPoint2[12766] = {X 275.5494, Y 92.7193, Z -3.0000, A 0.000, B 0.000, C 0.000 }
gfCNCPoint2[12767] = {X 275.5494, Y 85.6495, Z -3.0000, A 0.000, B 0.000, C 0.000 }
gfCNCPoint2[12768] = {X 262.6480, Y 80.5922, Z -3.0000, A 0.000, B 0.000, C 0.000 }
gfCNCPoint2[12769] = {X 262.3193, Y 80.7991, Z -3.0000, A 0.000, B 0.000, C 0.000 }
gfCNCPoint2[12770] = {X 237.8765, Y 96.6313, Z -3.0000, A 0.000, B 0.000, C 0.000 }
gfCNCPoint2[12771] = {X 237.8798, Y 97.0659, Z -3.0000, A 0.000, B 0.000, C 0.000 }
gfCNCPoint2[12772] = {X 237.8798, Y 98.0000, Z -3.0000, A 0.000, B 0.000, C 0.000 }
gfCNCPoint2[12773] = {X 237.7695, Y 98.9791, Z -3.0000, A 0.000, B 0.000, C 0.000 }
gfCNCPoint2[12774] = {X 237.4440, Y 99.9091, Z -3.0000, A 0.000, B 0.000, C 0.000 }
gfCNCPoint2[12775] = {X 236.9198, Y 100.7434, Z -3.0000, A 0.000, B 0.000, C 0.000 }
gfCNCPoint2[12776] = {X 236.2231, Y 101.4401, Z -3.0000, A 0.000, B 0.000, C 0.000 }
gfCNCPoint2[12777] = {X 235.3889, Y 101.9643, Z -3.0000, A 0.000, B 0.000, C 0.000 }
gfCNCPoint2[12778] = {X 234.4589, Y 102.2897, Z -3.0000, A 0.000, B 0.000, C 0.000 }
gfCNCPoint2[12779] = {X 233.4798, Y 102.4000, Z -3.0000, A 0.000, B 0.000, C 0.000 }
gfCNCPoint2[12780] = {X 214.1790, Y 102.4000, Z -3.0000, A 0.000, B 0.000, C 0.000 }
gfCNCPoint2[12781] = {X 213.7862, Y 102.3824, Z -3.0000, A 0.000, B 0.000, C 0.000 }
gfCNCPoint2[12782] = {X 213.3966, Y 102.3299, Z -3.0000, A 0.000, B 0.000, C 0.000 }
gfCNCPoint2[12783] = {X 213.0069, Y 102.3824, Z -3.0000, A 0.000, B 0.000, C 0.000 }
gfCNCPoint2[12784] = {X 212.6141, Y 102.4000, Z -3.0000, A 0.000, B 0.000, C 0.000 }
gfCNCPoint2[12785] = {X 194.9870, Y 102.4000, Z -3.0000, A 0.000, B 0.000, C 0.000 }
gfCNCPoint2[12786] = {X 194.0079, Y 102.2897, Z -3.0000, A 0.000, B 0.000, C 0.000 }
gfCNCPoint2[12787] = {X 193.0779, Y 101.9643, Z -3.0000, A 0.000, B 0.000, C 0.000 }
gfCNCPoint2[12788] = {X 192.2436, Y 101.4401, Z -3.0000, A 0.000, B 0.000, C 0.000 }
gfCNCPoint2[12789] = {X 191.5469, Y 100.7434, Z -3.0000, A 0.000, B 0.000, C 0.000 }
gfCNCPoint2[12790] = {X 191.0227, Y 99.9091, Z -3.0000, A 0.000, B 0.000, C 0.000 }
gfCNCPoint2[12791] = {X 190.6973, Y 98.9791, Z -3.0000, A 0.000, B 0.000, C 0.000 }
gfCNCPoint2[12792] = {X 190.5870, Y 98.0000, Z -3.0000, A 0.000, B 0.000, C 0.000 }
gfCNCPoint2[12793] = {X 190.5870, Y 97.0659, Z -3.0000, A 0.000, B 0.000, C 0.000 }
gfCNCPoint2[12794] = {X 190.6897, Y 96.1207, Z -3.0000, A 0.000, B 0.000, C 0.000 }
gfCNCPoint2[12795] = {X 190.9931, Y 95.2196, Z -3.0000, A 0.000, B 0.000, C 0.000 }
gfCNCPoint2[12796] = {X 191.4830, Y 94.4047, Z -3.0000, A 0.000, B 0.000, C 0.000 }
gfCNCPoint2[12797] = {X 188.5295, Y 91.1802, Z -3.0000, A 0.000, B 0.000, C 0.000 }
gfCNCPoint2[12798] = {X 150.1254, Y 91.1802, Z -3.0000, A 0.000, B 0.000, C 0.000 }
gfCNCPoint2[12799] = {X 147.2493, Y 94.3666, Z -3.0000, A 0.000, B 0.000, C 0.000 }
gfCNCPoint2[12800] = {X 147.7552, Y 95.1908, Z -3.0000, A 0.000, B 0.000, C 0.000 }
gfCNCPoint2[12801] = {X 148.0701, Y 96.1052, Z -3.0000, A 0.000, B 0.000, C 0.000 }
gfCNCPoint2[12802] = {X 148.1791, Y 97.0661, Z -3.0000, A 0.000, B 0.000, C 0.000 }
gfCNCPoint2[12803] = {X 148.1791, Y 98.0000, Z -3.0000, A 0.000, B 0.000, C 0.000 }
gfCNCPoint2[12804] = {X 148.0688, Y 98.9791, Z -3.0000, A 0.000, B 0.000, C 0.000 }
gfCNCPoint2[12805] = {X 147.7434, Y 99.9091, Z -3.0000, A 0.000, B 0.000, C 0.000 }
gfCNCPoint2[12806] = {X 147.2192, Y 100.7434, Z -3.0000, A 0.000, B 0.000, C 0.000 }
gfCNCPoint2[12807] = {X 146.5225, Y 101.4401, Z -3.0000, A 0.000, B 0.000, C 0.000 }
gfCNCPoint2[12808] = {X 145.6882, Y 101.9643, Z -3.0000, A 0.000, B 0.000, C 0.000 }
gfCNCPoint2[12809] = {X 144.7582, Y 102.2897, Z -3.0000, A 0.000, B 0.000, C 0.000 }
gfCNCPoint2[12810] = {X 143.7791, Y 102.4000, Z -3.0000, A 0.000, B 0.000, C 0.000 }
gfCNCPoint2[12811] = {X 125.0000, Y 102.4000, Z -3.0000, A 0.000, B 0.000, C 0.000 }
gfCNCPoint2[12812] = {X 124.0209, Y 102.2897, Z -3.0000, A 0.000, B 0.000, C 0.000 }
gfCNCPoint2[12813] = {X 123.0909, Y 101.9643, Z -3.0000, A 0.000, B 0.000, C 0.000 }
gfCNCPoint2[12814] = {X 122.2566, Y 101.4401, Z -3.0000, A 0.000, B 0.000, C 0.000 }
gfCNCPoint2[12815] = {X 121.5599, Y 100.7434, Z -3.0000, A 0.000, B 0.000, C 0.000 }
gfCNCPoint2[12816] = {X 121.0357, Y 99.9091, Z -3.0000, A 0.000, B 0.000, C 0.000 }
gfCNCPoint2[12817] = {X 120.7103, Y 98.9791, Z -3.0000, A 0.000, B 0.000, C 0.000 }
gfCNCPoint2[12818] = {X 120.6000, Y 98.0000, Z -3.0000, A 0.000, B 0.000, C 0.000 }
gfCNCPoint2[12819] = {X 120.6000, Y 97.0659, Z -3.0000, A 0.000, B 0.000, C 0.000 }
gfCNCPoint2[12820] = {X 120.7047, Y 96.1118, Z -3.0000, A 0.000, B 0.000, C 0.000 }
gfCNCPoint2[12821] = {X 121.0138, Y 95.2031, Z -3.0000, A 0.000, B 0.000, C 0.000 }
gfCNCPoint2[12822] = {X 121.5125, Y 94.3831, Z -3.0000, A 0.000, B 0.000, C 0.000 }
gfCNCPoint2[12823] = {X 122.1773, Y 93.6907, Z -3.0000, A 0.000, B 0.000, C 0.000 }
gfCNCPoint2[12824] = {X 122.9763, Y 93.1589, Z -3.0000, A 0.000, B 0.000, C 0.000 }
gfCNCPoint2[12825] = {X 123.8716, Y 92.8131, Z -3.0000, A 0.000, B 0.000, C 0.000 }
gfCNCPoint2[12826] = {X 124.8207, Y 92.6696, Z -3.0000, A 0.000, B 0.000, C 0.000 }
gfCNCPoint2[12827] = {X 124.8676, Y 92.6533, Z -3.0000, A 0.000, B 0.000, C 0.000 }
gfCNCPoint2[12828] = {X 124.9162, Y 92.6430, Z -3.0000, A 0.000, B 0.000, C 0.000 }
gfCNCPoint2[12829] = {X 125.4406, Y 92.5652, Z -3.0000, A 0.000, B 0.000, C 0.000 }
gfCNCPoint2[12830] = {X 126.2564, Y 92.4276, Z -3.0000, A 0.000, B 0.000, C 0.000 }
gfCNCPoint2[12831] = {X 127.0613, Y 92.2361, Z -3.0000, A 0.000, B 0.000, C 0.000 }
gfCNCPoint2[12832] = {X 128.2731, Y 91.0926, Z -3.0000, A 0.000, B 0.000, C 0.000 }
gfCNCPoint2[12833] = {X 129.4213, Y 89.8854, Z -3.0000, A 0.000, B 0.000, C 0.000 }
gfCNCPoint2[12834] = {X 133.5081, Y 85.3898, Z -3.0000, A 0.000, B 0.000, C 0.000 }
gfCNCPoint2[12835] = {X 155.5330, Y 61.2112, Z -3.0000, A 0.000, B 0.000, C 0.000 }
gfCNCPoint2[12836] = {X 155.1841, Y 60.4949, Z -3.0000, A 0.000, B 0.000, C 0.000 }
gfCNCPoint2[12837] = {X 154.9701, Y 59.7275, Z -3.0000, A 0.000, B 0.000, C 0.000 }
gfCNCPoint2[12838] = {X 154.8980, Y 58.9340, Z -3.0000, A 0.000, B 0.000, C 0.000 }
gfCNCPoint2[12839] = {X 154.8980, Y 58.0000, Z -3.0000, A 0.000, B 0.000, C 0.000 }
gfCNCPoint2[12840] = {X 155.0083, Y 57.0209, Z -3.0000, A 0.000, B 0.000, C 0.000 }
gfCNCPoint2[12841] = {X 155.3337, Y 56.0909, Z -3.0000, A 0.000, B 0.000, C 0.000 }
gfCNCPoint2[12842] = {X 155.8579, Y 55.2566, Z -3.0000, A 0.000, B 0.000, C 0.000 }
gfCNCPoint2[12843] = {X 156.5546, Y 54.5599, Z -3.0000, A 0.000, B 0.000, C 0.000 }
gfCNCPoint2[12844] = {X 157.3889, Y 54.0357, Z -3.0000, A 0.000, B 0.000, C 0.000 }
gfCNCPoint2[12845] = {X 158.3189, Y 53.7103, Z -3.0000, A 0.000, B 0.000, C 0.000 }
gfCNCPoint2[12846] = {X 159.2980, Y 53.6000, Z -3.0000, A 0.000, B 0.000, C 0.000 }
gfCNCPoint2[12847] = {X 178.5335, Y 53.6000, Z -3.0000, A 0.000, B 0.000, C 0.000 }
gfCNCPoint2[12848] = {X 179.5126, Y 53.7103, Z -3.0000, A 0.000, B 0.000, C 0.000 }
gfCNCPoint2[12849] = {X 180.4426, Y 54.0357, Z -3.0000, A 0.000, B 0.000, C 0.000 }
gfCNCPoint2[12850] = {X 181.2769, Y 54.5599, Z -3.0000, A 0.000, B 0.000, C 0.000 }
gfCNCPoint2[12851] = {X 181.9736, Y 55.2566, Z -3.0000, A 0.000, B 0.000, C 0.000 }
gfCNCPoint2[12852] = {X 182.4978, Y 56.0909, Z -3.0000, A 0.000, B 0.000, C 0.000 }
gfCNCPoint2[12853] = {X 182.8232, Y 57.0209, Z -3.0000, A 0.000, B 0.000, C 0.000 }
gfCNCPoint2[12854] = {X 182.9335, Y 58.0000, Z -3.0000, A 0.000, B 0.000, C 0.000 }
gfCNCPoint2[12855] = {X 182.9334, Y 58.9704, Z -3.0000, A 0.000, B 0.000, C 0.000 }
gfCNCPoint2[12856] = {X 182.8587, Y 59.7420, Z -3.0000, A 0.000, B 0.000, C 0.000 }
gfCNCPoint2[12857] = {X 182.6498, Y 60.4885, Z -3.0000, A 0.000, B 0.000, C 0.000 }
gfCNCPoint2[12858] = {X 182.3131, Y 61.1867, Z -3.0000, A 0.000, B 0.000, C 0.000 }
gfCNCPoint2[12859] = {X 209.5369, Y 90.8999, Z -3.0000, A 0.000, B 0.000, C 0.000 }
gfCNCPoint2[12860] = {X 210.1906, Y 91.5632, Z -3.0000, A 0.000, B 0.000, C 0.000 }
gfCNCPoint2[12861] = {X 210.8909, Y 92.1770, Z -3.0000, A 0.000, B 0.000, C 0.000 }
gfCNCPoint2[12862] = {X 211.1524, Y 92.3419, Z -3.0000, A 0.000, B 0.000, C 0.000 }
gfCNCPoint2[12863] = {X 211.4457, Y 92.4393, Z -3.0000, A 0.000, B 0.000, C 0.000 }
gfCNCPoint2[12864] = {X 212.1215, Y 92.5838, Z -3.0000, A 0.000, B 0.000, C 0.000 }
gfCNCPoint2[12865] = {X 213.4014, Y 92.7451, Z -3.0000, A 0.000, B 0.000, C 0.000 }
gfCNCPoint2[12866] = {X 214.4546, Y 92.6563, Z -3.0000, A 0.000, B 0.000, C 0.000 }
gfCNCPoint2[12867] = {X 215.5099, Y 92.5962, Z -3.0000, A 0.000, B 0.000, C 0.000 }
gfCNCPoint2[12868] = {X 216.1639, Y 92.5240, Z -3.0000, A 0.000, B 0.000, C 0.000 }
gfCNCPoint2[12869] = {X 216.7937, Y 92.3333, Z -3.0000, A 0.000, B 0.000, C 0.000 }
gfCNCPoint2[12870] = {X 217.3778, Y 92.0304, Z -3.0000, A 0.000, B 0.000, C 0.000 }
gfCNCPoint2[12871] = {X 222.9188, Y 88.4545, Z -3.0000, A 0.000, B 0.000, C 0.000 }
gfCNCPoint2[12872] = {X 245.6535, Y 73.9166, Z -3.0000, A 0.000, B 0.000, C 0.000 }
gfCNCPoint2[12873] = {X 221.6008, Y 64.4773, Z -3.0000, A 0.000, B 0.000, C 0.000 }
gfCNCPoint2[12874] = {X 219.8423, Y 63.8888, Z -3.0000, A 0.000, B 0.000, C 0.000 }
gfCNCPoint2[12875] = {X 218.0280, Y 63.5052, Z -3.0000, A 0.000, B 0.000, C 0.000 }
gfCNCPoint2[12876] = {X 216.1817, Y 63.3315, Z -3.0000, A 0.000, B 0.000, C 0.000 }
gfCNCPoint2[12877] = {X 215.2275, Y 63.1935, Z -3.0000, A 0.000, B 0.000, C 0.000 }
gfCNCPoint2[12878] = {X 214.3263, Y 62.8509, Z -3.0000, A 0.000, B 0.000, C 0.000 }
gfCNCPoint2[12879] = {X 213.5213, Y 62.3203, Z -3.0000, A 0.000, B 0.000, C 0.000 }
gfCNCPoint2[12880] = {X 212.8512, Y 61.6271, Z -3.0000, A 0.000, B 0.000, C 0.000 }
gfCNCPoint2[12881] = {X 212.3482, Y 60.8047, Z -3.0000, A 0.000, B 0.000, C 0.000 }
gfCNCPoint2[12882] = {X 212.0364, Y 59.8924, Z -3.0000, A 0.000, B 0.000, C 0.000 }
gfCNCPoint2[12883] = {X 211.9308, Y 58.9340, Z -3.0000, A 0.000, B 0.000, C 0.000 }
gfCNCPoint2[12884] = {X 211.9308, Y 58.0000, Z -3.0000, A 0.000, B 0.000, C 0.000 }
gfCNCPoint2[12885] = {X 212.0411, Y 57.0209, Z -3.0000, A 0.000, B 0.000, C 0.000 }
gfCNCPoint2[12886] = {X 212.3665, Y 56.0909, Z -3.0000, A 0.000, B 0.000, C 0.000 }
gfCNCPoint2[12887] = {X 212.8907, Y 55.2566, Z -3.0000, A 0.000, B 0.000, C 0.000 }
gfCNCPoint2[12888] = {X 213.5875, Y 54.5599, Z -3.0000, A 0.000, B 0.000, C 0.000 }
gfCNCPoint2[12889] = {X 214.4217, Y 54.0357, Z -3.0000, A 0.000, B 0.000, C 0.000 }
gfCNCPoint2[12890] = {X 215.3517, Y 53.7103, Z -3.0000, A 0.000, B 0.000, C 0.000 }
gfCNCPoint2[12891] = {X 216.3308, Y 53.6000, Z -3.0000, A 0.000, B 0.000, C 0.000 }
gfCNCPoint2[12892] = {X 237.2617, Y 53.6000, Z -3.0000, A 0.000, B 0.000, C 0.000 }
gfCNCPoint2[12893] = {X 238.2408, Y 53.7103, Z -3.0000, A 0.000, B 0.000, C 0.000 }
gfCNCPoint2[12894] = {X 239.1708, Y 54.0357, Z -3.0000, A 0.000, B 0.000, C 0.000 }
gfCNCPoint2[12895] = {X 240.0050, Y 54.5599, Z -3.0000, A 0.000, B 0.000, C 0.000 }
gfCNCPoint2[12896] = {X 240.7017, Y 55.2566, Z -3.0000, A 0.000, B 0.000, C 0.000 }
gfCNCPoint2[12897] = {X 241.2260, Y 56.0909, Z -3.0000, A 0.000, B 0.000, C 0.000 }
gfCNCPoint2[12898] = {X 241.5514, Y 57.0209, Z -3.0000, A 0.000, B 0.000, C 0.000 }
gfCNCPoint2[12899] = {X 241.6617, Y 58.0000, Z -3.0000, A 0.000, B 0.000, C 0.000 }
gfCNCPoint2[12900] = {X 241.6617, Y 58.1780, Z -3.0000, A 0.000, B 0.000, C 0.000 }
gfCNCPoint2[12901] = {X 247.5187, Y 60.4613, Z -3.0000, A 0.000, B 0.000, C 0.000 }
gfCNCPoint2[12902] = {X 275.5534, Y 71.5849, Z -3.0000, A 0.000, B 0.000, C 0.000 }
gfCNCPoint2[12903] = {X 275.5528, Y 63.2812, Z -3.0000, A 0.000, B 0.000, C 0.000 }
gfCNCPoint2[12904] = {X 274.6935, Y 63.0561, Z -3.0000, A 0.000, B 0.000, C 0.000 }
gfCNCPoint2[12905] = {X 273.8969, Y 62.6629, Z -3.0000, A 0.000, B 0.000, C 0.000 }
gfCNCPoint2[12906] = {X 273.1955, Y 62.1177, Z -3.0000, A 0.000, B 0.000, C 0.000 }
gfCNCPoint2[12907] = {X 272.6180, Y 61.4428, Z -3.0000, A 0.000, B 0.000, C 0.000 }
gfCNCPoint2[12908] = {X 272.1877, Y 60.6656, Z -3.0000, A 0.000, B 0.000, C 0.000 }
gfCNCPoint2[12909] = {X 271.9224, Y 59.8178, Z -3.0000, A 0.000, B 0.000, C 0.000 }
gfCNCPoint2[12910] = {X 271.8327, Y 58.9340, Z -3.0000, A 0.000, B 0.000, C 0.000 }
gfCNCPoint2[12911] = {X 271.8327, Y 58.0000, Z -3.0000, A 0.000, B 0.000, C 0.000 }
gfCNCPoint2[12912] = {X 271.9430, Y 57.0209, Z -3.0000, A 0.000, B 0.000, C 0.000 }
gfCNCPoint2[12913] = {X 272.2684, Y 56.0909, Z -3.0000, A 0.000, B 0.000, C 0.000 }
gfCNCPoint2[12914] = {X 272.7926, Y 55.2566, Z -3.0000, A 0.000, B 0.000, C 0.000 }
gfCNCPoint2[12915] = {X 273.4893, Y 54.5599, Z -3.0000, A 0.000, B 0.000, C 0.000 }
gfCNCPoint2[12916] = {X 274.3236, Y 54.0357, Z -3.0000, A 0.000, B 0.000, C 0.000 }
gfCNCPoint2[12917] = {X 275.2536, Y 53.7103, Z -3.0000, A 0.000, B 0.000, C 0.000 }
gfCNCPoint2[12918] = {X 276.2327, Y 53.6000, Z -3.0000, A 0.000, B 0.000, C 0.000 }
gfCNCPoint2[12919] = {X 292.7731, Y 53.6000, Z -3.0000, A 0.000, B 0.000, C 0.000 }
gfCNCPoint2[12920] = {X 293.7522, Y 53.7103, Z -3.0000, A 0.000, B 0.000, C 0.000 }
gfCNCPoint2[12921] = {X 294.6822, Y 54.0357, Z -3.0000, A 0.000, B 0.000, C 0.000 }
gfCNCPoint2[12922] = {X 295.5164, Y 54.5599, Z -3.0000, A 0.000, B 0.000, C 0.000 }
gfCNCPoint2[12923] = {X 296.2131, Y 55.2566, Z -3.0000, A 0.000, B 0.000, C 0.000 }
gfCNCPoint2[12924] = {X 296.7373, Y 56.0909, Z -3.0000, A 0.000, B 0.000, C 0.000 }
gfCNCPoint2[12925] = {X 297.0628, Y 57.0209, Z -3.0000, A 0.000, B 0.000, C 0.000 }
gfCNCPoint2[12926] = {X 297.1731, Y 58.0000, Z -3.0000, A 0.000, B 0.000, C 0.000 }
gfCNCPoint2[12927] = {X 297.1731, Y 58.9354, Z -3.0000, A 0.000, B 0.000, C 0.000 }
gfCNCPoint2[12928] = {X 297.0809, Y 59.8183, Z -3.0000, A 0.000, B 0.000, C 0.000 }
gfCNCPoint2[12929] = {X 296.8141, Y 60.6650, Z -3.0000, A 0.000, B 0.000, C 0.000 }
gfCNCPoint2[12930] = {X 296.3833, Y 61.4412, Z -3.0000, A 0.000, B 0.000, C 0.000 }
gfCNCPoint2[12931] = {X 295.8060, Y 62.1155, Z -3.0000, A 0.000, B 0.000, C 0.000 }
gfCNCPoint2[12932] = {X 295.1056, Y 62.6608, Z -3.0000, A 0.000, B 0.000, C 0.000 }
gfCNCPoint2[12933] = {X 294.3102, Y 63.0551, Z -3.0000, A 0.000, B 0.000, C 0.000 }
gfCNCPoint2[12934] = {X 293.4521, Y 63.2823, Z -3.0000, A 0.000, B 0.000, C 0.000 }
gfCNCPoint2[12935] = {X 293.4521, Y 92.7114, Z -3.0000, A 0.000, B 0.000, C 0.000 }
gfCNCPoint2[12936] = {X 294.3100, Y 92.9411, Z -3.0000, A 0.000, B 0.000, C 0.000 }
gfCNCPoint2[12937] = {X 295.1049, Y 93.3373, Z -3.0000, A 0.000, B 0.000, C 0.000 }
gfCNCPoint2[12938] = {X 295.8049, Y 93.8839, Z -3.0000, A 0.000, B 0.000, C 0.000 }
gfCNCPoint2[12939] = {X 296.3819, Y 94.5592, Z -3.0000, A 0.000, B 0.000, C 0.000 }
gfCNCPoint2[12940] = {X 296.8127, Y 95.3359, Z -3.0000, A 0.000, B 0.000, C 0.000 }
gfCNCPoint2[12941] = {X 297.0800, Y 96.1828, Z -3.0000, A 0.000, B 0.000, C 0.000 }
gfCNCPoint2[12942] = {X 297.1731, Y 97.0661, Z -3.0000, A 0.000, B 0.000, C 0.000 }
gfCNCPoint2[12943] = {X 297.1731, Y 97.6950, Z -3.0000, A 0.000, B 0.000, C 0.000 }
gfCNCPoint2[12944] = {X 297.6531, Y 97.6950, Z -3.0000, A 0.000, B 0.000, C 0.000 }
gfCNCPoint2[12945] = {X 314.2153, Y 97.6950, Z -3.0000, A 0.000, B 0.000, C 0.000 }
gfCNCPoint2[12946] = {X 313.0165, Y 96.8442, Z -3.0000, A 0.000, B 0.000, C 0.000 }
gfCNCPoint2[12947] = {X 311.8816, Y 95.9098, Z -3.0000, A 0.000, B 0.000, C 0.000 }
gfCNCPoint2[12948] = {X 310.9060, Y 94.9482, Z -3.0000, A 0.000, B 0.000, C 0.000 }
gfCNCPoint2[12949] = {X 310.0418, Y 93.8854, Z -3.0000, A 0.000, B 0.000, C 0.000 }
gfCNCPoint2[12950] = {X 309.2078, Y 92.5707, Z -3.0000, A 0.000, B 0.000, C 0.000 }
gfCNCPoint2[12951] = {X 308.5442, Y 91.1624, Z -3.0000, A 0.000, B 0.000, C 0.000 }
gfCNCPoint2[12952] = {X 308.0611, Y 89.6824, Z -3.0000, A 0.000, B 0.000, C 0.000 }
gfCNCPoint2[12953] = {X 307.7077, Y 88.0125, Z -3.0000, A 0.000, B 0.000, C 0.000 }
gfCNCPoint2[12954] = {X 307.4988, Y 86.3184, Z -3.0000, A 0.000, B 0.000, C 0.000 }
gfCNCPoint2[12955] = {X 307.4360, Y 84.6126, Z -3.0000, A 0.000, B 0.000, C 0.000 }
gfCNCPoint2[12956] = {X 307.4373, Y 83.2305, Z -3.0000, A 0.000, B 0.000, C 0.000 }
gfCNCPoint2[12957] = {X 307.4373, Y 63.6745, Z -3.0000, A 0.000, B 0.000, C 0.000 }
gfCNCPoint2[12958] = {X 306.4287, Y 63.3063, Z -3.0000, A 0.000, B 0.000, C 0.000 }
gfCNCPoint2[12959] = {X 305.5251, Y 62.7265, Z -3.0000, A 0.000, B 0.000, C 0.000 }
gfCNCPoint2[12960] = {X 304.7701, Y 61.9631, Z -3.0000, A 0.000, B 0.000, C 0.000 }
gfCNCPoint2[12961] = {X 304.2003, Y 61.0531, Z -3.0000, A 0.000, B 0.000, C 0.000 }
gfCNCPoint2[12962] = {X 303.8433, Y 60.0405, Z -3.0000, A 0.000, B 0.000, C 0.000 }
gfCNCPoint2[12963] = {X 303.7164, Y 58.9744, Z -3.0000, A 0.000, B 0.000, C 0.000 }
gfCNCPoint2[12964] = {X 303.7162, Y 58.0000, Z -3.0000, A 0.000, B 0.000, C 0.000 }
gfCNCPoint2[12965] = {X 303.8100, Y 57.0480, Z -3.0000, A 0.000, B 0.000, C 0.000 }
gfCNCPoint2[12966] = {X 304.0877, Y 56.1325, Z -3.0000, A 0.000, B 0.000, C 0.000 }
gfCNCPoint2[12967] = {X 304.5387, Y 55.2888, Z -3.0000, A 0.000, B 0.000, C 0.000 }
gfCNCPoint2[12968] = {X 305.1455, Y 54.5493, Z -3.0000, A 0.000, B 0.000, C 0.000 }
gfCNCPoint2[12969] = {X 305.8850, Y 53.9424, Z -3.0000, A 0.000, B 0.000, C 0.000 }
gfCNCPoint2[12970] = {X 306.7287, Y 53.4915, Z -3.0000, A 0.000, B 0.000, C 0.000 }
gfCNCPoint2[12971] = {X 307.6442, Y 53.2138, Z -3.0000, A 0.000, B 0.000, C 0.000 }
gfCNCPoint2[12972] = {X 308.5962, Y 53.1200, Z -3.0000, A 0.000, B 0.000, C 0.000 }
gfCNCPoint2[12973] = {X 324.3107, Y 53.1200, Z -3.0000, A 0.000, B 0.000, C 0.000 }
gfCNCPoint2[12974] = {X 325.2627, Y 53.2138, Z -3.0000, A 0.000, B 0.000, C 0.000 }
gfCNCPoint2[12975] = {X 326.1782, Y 53.4915, Z -3.0000, A 0.000, B 0.000, C 0.000 }
gfCNCPoint2[12976] = {X 327.0219, Y 53.9424, Z -3.0000, A 0.000, B 0.000, C 0.000 }
gfCNCPoint2[12977] = {X 327.7614, Y 54.5493, Z -3.0000, A 0.000, B 0.000, C 0.000 }
gfCNCPoint2[12978] = {X 328.3683, Y 55.2888, Z -3.0000, A 0.000, B 0.000, C 0.000 }
gfCNCPoint2[12979] = {X 328.8192, Y 56.1325, Z -3.0000, A 0.000, B 0.000, C 0.000 }
gfCNCPoint2[12980] = {X 329.0969, Y 57.0480, Z -3.0000, A 0.000, B 0.000, C 0.000 }
gfCNCPoint2[12981] = {X 329.1907, Y 58.0000, Z -3.0000, A 0.000, B 0.000, C 0.000 }
gfCNCPoint2[12982] = {X 329.1907, Y 58.9341, Z -3.0000, A 0.000, B 0.000, C 0.000 }
gfCNCPoint2[12983] = {X 329.0669, Y 60.0066, Z -3.0000, A 0.000, B 0.000, C 0.000 }
gfCNCPoint2[12984] = {X 328.7121, Y 61.0263, Z -3.0000, A 0.000, B 0.000, C 0.000 }
gfCNCPoint2[12985] = {X 328.1435, Y 61.9441, Z -3.0000, A 0.000, B 0.000, C 0.000 }
gfCNCPoint2[12986] = {X 327.3883, Y 62.7157, Z -3.0000, A 0.000, B 0.000, C 0.000 }
gfCNCPoint2[12987] = {X 326.4829, Y 63.3040, Z -3.0000, A 0.000, B 0.000, C 0.000 }
gfCNCPoint2[12988] = {X 325.4711, Y 63.6806, Z -3.0000, A 0.000, B 0.000, C 0.000 }
gfCNCPoint2[12989] = {X 325.4726, Y 83.2268, Z -3.0000, A 0.000, B 0.000, C 0.000 }
gfCNCPoint2[12990] = {X 325.4861, Y 84.6073, Z -3.0000, A 0.000, B 0.000, C 0.000 }
gfCNCPoint2[12991] = {X 325.5519, Y 85.7202, Z -3.0000, A 0.000, B 0.000, C 0.000 }
gfCNCPoint2[12992] = {X 325.7424, Y 86.8186, Z -3.0000, A 0.000, B 0.000, C 0.000 }
gfCNCPoint2[12993] = {X 325.8863, Y 86.9528, Z -3.0000, A 0.000, B 0.000, C 0.000 }
gfCNCPoint2[12994] = {X 326.0546, Y 87.0550, Z -3.0000, A 0.000, B 0.000, C 0.000 }
gfCNCPoint2[12995] = {X 326.4832, Y 87.2971, Z -3.0000, A 0.000, B 0.000, C 0.000 }
gfCNCPoint2[12996] = {X 327.8564, Y 87.8659, Z -3.0000, A 0.000, B 0.000, C 0.000 }
gfCNCPoint2[12997] = {X 329.2835, Y 88.2812, Z -3.0000, A 0.000, B 0.000, C 0.000 }
gfCNCPoint2[12998] = {X 332.3214, Y 88.8896, Z -3.0000, A 0.000, B 0.000, C 0.000 }
gfCNCPoint2[12999] = {X 335.3953, Y 89.2774, Z -3.0000, A 0.000, B 0.000, C 0.000 }
gfCNCPoint2[13000] = {X 339.5149, Y 89.5966, Z -3.0000, A 0.000, B 0.000, C 0.000 }
gfCNCPoint2[13001] = {X 343.6429, Y 89.7756, Z -3.0000, A 0.000, B 0.000, C 0.000 }
gfCNCPoint2[13002] = {X 347.7746, Y 89.8141, Z -3.0000, A 0.000, B 0.000, C 0.000 }
gfCNCPoint2[13003] = {X 352.1398, Y 89.7761, Z -3.0000, A 0.000, B 0.000, C 0.000 }
gfCNCPoint2[13004] = {X 356.5008, Y 89.5811, Z -3.0000, A 0.000, B 0.000, C 0.000 }
gfCNCPoint2[13005] = {X 360.8519, Y 89.2294, Z -3.0000, A 0.000, B 0.000, C 0.000 }
gfCNCPoint2[13006] = {X 363.1336, Y 88.9458, Z -3.0000, A 0.000, B 0.000, C 0.000 }
gfCNCPoint2[13007] = {X 365.3941, Y 88.5255, Z -3.0000, A 0.000, B 0.000, C 0.000 }
gfCNCPoint2[13008] = {X 367.6252, Y 87.9700, Z -3.0000, A 0.000, B 0.000, C 0.000 }
gfCNCPoint2[13009] = {X 368.9189, Y 87.4951, Z -3.0000, A 0.000, B 0.000, C 0.000 }
gfCNCPoint2[13010] = {X 370.1146, Y 86.8100, Z -3.0000, A 0.000, B 0.000, C 0.000 }
gfCNCPoint2[13011] = {X 370.2992, Y 85.3241, Z -3.0000, A 0.000, B 0.000, C 0.000 }
gfCNCPoint2[13012] = {X 370.3608, Y 83.8280, Z -3.0000, A 0.000, B 0.000, C 0.000 }
gfCNCPoint2[13013] = {X 370.3592, Y 63.6742, Z -3.0000, A 0.000, B 0.000, C 0.000 }
gfCNCPoint2[13014] = {X 369.3509, Y 63.3058, Z -3.0000, A 0.000, B 0.000, C 0.000 }
gfCNCPoint2[13015] = {X 368.4475, Y 62.7260, Z -3.0000, A 0.000, B 0.000, C 0.000 }
gfCNCPoint2[13016] = {X 367.6928, Y 61.9626, Z -3.0000, A 0.000, B 0.000, C 0.000 }
gfCNCPoint2[13017] = {X 367.1232, Y 61.0527, Z -3.0000, A 0.000, B 0.000, C 0.000 }
gfCNCPoint2[13018] = {X 366.7663, Y 60.0403, Z -3.0000, A 0.000, B 0.000, C 0.000 }
gfCNCPoint2[13019] = {X 366.6394, Y 58.9744, Z -3.0000, A 0.000, B 0.000, C 0.000 }
gfCNCPoint2[13020] = {X 366.6393, Y 58.0000, Z -3.0000, A 0.000, B 0.000, C 0.000 }
gfCNCPoint2[13021] = {X 366.7331, Y 57.0480, Z -3.0000, A 0.000, B 0.000, C 0.000 }
gfCNCPoint2[13022] = {X 367.0108, Y 56.1325, Z -3.0000, A 0.000, B 0.000, C 0.000 }
gfCNCPoint2[13023] = {X 367.4617, Y 55.2888, Z -3.0000, A 0.000, B 0.000, C 0.000 }
gfCNCPoint2[13024] = {X 368.0686, Y 54.5493, Z -3.0000, A 0.000, B 0.000, C 0.000 }
gfCNCPoint2[13025] = {X 368.8081, Y 53.9424, Z -3.0000, A 0.000, B 0.000, C 0.000 }
gfCNCPoint2[13026] = {X 369.6518, Y 53.4915, Z -3.0000, A 0.000, B 0.000, C 0.000 }
gfCNCPoint2[13027] = {X 370.5672, Y 53.2138, Z -3.0000, A 0.000, B 0.000, C 0.000 }
gfCNCPoint2[13028] = {X 371.5193, Y 53.1200, Z -3.0000, A 0.000, B 0.000, C 0.000 }
gfCNCPoint2[13029] = {X 388.0597, Y 53.1200, Z -3.0000, A 0.000, B 0.000, C 0.000 }
gfCNCPoint2[13030] = {X 389.0355, Y 53.2186, Z -3.0000, A 0.000, B 0.000, C 0.000 }
gfCNCPoint2[13031] = {X 389.9719, Y 53.5102, Z -3.0000, A 0.000, B 0.000, C 0.000 }
gfCNCPoint2[13032] = {X 390.8310, Y 53.9833, Z -3.0000, A 0.000, B 0.000, C 0.000 }
gfCNCPoint2[13033] = {X 391.5783, Y 54.6186, Z -3.0000, A 0.000, B 0.000, C 0.000 }
gfCNCPoint2[13034] = {X 392.1572, Y 55.3496, Z -3.0000, A 0.000, B 0.000, C 0.000 }
gfCNCPoint2[13035] = {X 392.5865, Y 56.1774, Z -3.0000, A 0.000, B 0.000, C 0.000 }
gfCNCPoint2[13036] = {X 392.8506, Y 57.0718, Z -3.0000, A 0.000, B 0.000, C 0.000 }
gfCNCPoint2[13037] = {X 392.9397, Y 58.0000, Z -3.0000, A 0.000, B 0.000, C 0.000 }
gfCNCPoint2[13038] = {X 392.9395, Y 58.9744, Z -3.0000, A 0.000, B 0.000, C 0.000 }
gfCNCPoint2[13039] = {X 392.8775, Y 59.7105, Z -3.0000, A 0.000, B 0.000, C 0.000 }
gfCNCPoint2[13040] = {X 392.7051, Y 60.4288, Z -3.0000, A 0.000, B 0.000, C 0.000 }
gfCNCPoint2[13041] = {X 392.4263, Y 61.1129, Z -3.0000, A 0.000, B 0.000, C 0.000 }
gfCNCPoint2[13042] = {X 392.0474, Y 61.7474, Z -3.0000, A 0.000, B 0.000, C 0.000 }
gfCNCPoint2[13043] = {X 391.5775, Y 62.3177, Z -3.0000, A 0.000, B 0.000, C 0.000 }
gfCNCPoint2[13044] = {X 390.8817, Y 62.9184, Z -3.0000, A 0.000, B 0.000, C 0.000 }
gfCNCPoint2[13045] = {X 390.0860, Y 63.3787, Z -3.0000, A 0.000, B 0.000, C 0.000 }
gfCNCPoint2[13046] = {X 389.2183, Y 63.6823, Z -3.0000, A 0.000, B 0.000, C 0.000 }
gfCNCPoint2[13047] = {X 389.2174, Y 73.4809, Z -3.0000, A 0.000, B 0.000, C 0.000 }
gfCNCPoint2[13048] = {X 398.8174, Y 73.4818, Z -3.0000, A 0.000, B 0.000, C 0.000 }
gfCNCPoint2[13049] = {X 398.8167, Y 80.5588, Z -3.0000, A 0.000, B 0.000, C 0.000 }
gfCNCPoint2[13050] = {X 405.8048, Y 76.0833, Z -3.0000, A 0.000, B 0.000, C 0.000 }
gfCNCPoint2[13051] = {X 400.0361, Y 73.8199, Z -3.0000, A 0.000, B 0.000, C 0.000 }
gfCNCPoint2[13052] = {X 399.4355, Y 73.6191, Z -3.0000, A 0.000, B 0.000, C 0.000 }
gfCNCPoint2[13053] = {X 398.8174, Y 73.4818, Z -3.0000, A 0.000, B 0.000, C 0.000 }
gfCNCPoint2[13054] = {X 396.4174, Y 73.4816, Z -3.0000, A 0.000, B 0.000, C 0.000 }
gfCNCPoint2[13055] = {X 396.4163, Y 84.5893, Z -3.0000, A 0.000, B 0.000, C 0.000 }
gfCNCPoint2[13056] = {X 396.4162, Y 84.9462, Z -3.0000, A 0.000, B 0.000, C 0.000 }
gfCNCPoint2[13057] = {X 411.0605, Y 75.5673, Z -3.0000, A 0.000, B 0.000, C 0.000 }
gfCNCPoint2[13058] = {X 400.9148, Y 71.5865, Z -3.0000, A 0.000, B 0.000, C 0.000 }
gfCNCPoint2[13059] = {X 399.6208, Y 71.1933, Z -3.0000, A 0.000, B 0.000, C 0.000 }
gfCNCPoint2[13060] = {X 398.2807, Y 71.0109, Z -3.0000, A 0.000, B 0.000, C 0.000 }
gfCNCPoint2[13061] = {X 397.3455, Y 70.9531, Z -3.0000, A 0.000, B 0.000, C 0.000 }
gfCNCPoint2[13062] = {X 396.4176, Y 70.8230, Z -3.0000, A 0.000, B 0.000, C 0.000 }
gfCNCPoint2[13063] = {X 396.4174, Y 73.4816, Z -3.0000, A 0.000, B 0.000, C 0.000 }
gfCNCPoint2[13064] = {X 394.0174, Y 73.4813, Z -3.0000, A 0.000, B 0.000, C 0.000 }
gfCNCPoint2[13065] = {X 394.0163, Y 84.5970, Z -3.0000, A 0.000, B 0.000, C 0.000 }
gfCNCPoint2[13066] = {X 394.0168, Y 84.7633, Z -3.0000, A 0.000, B 0.000, C 0.000 }
gfCNCPoint2[13067] = {X 394.0162, Y 84.9296, Z -3.0000, A 0.000, B 0.000, C 0.000 }
gfCNCPoint2[13068] = {X 393.9659, Y 86.3343, Z -3.0000, A 0.000, B 0.000, C 0.000 }
gfCNCPoint2[13069] = {X 393.8346, Y 87.7337, Z -3.0000, A 0.000, B 0.000, C 0.000 }
gfCNCPoint2[13070] = {X 395.0689, Y 87.4787, Z -3.0000, A 0.000, B 0.000, C 0.000 }
gfCNCPoint2[13071] = {X 396.3259, Y 87.3863, Z -3.0000, A 0.000, B 0.000, C 0.000 }
gfCNCPoint2[13072] = {X 396.7218, Y 87.3729, Z -3.0000, A 0.000, B 0.000, C 0.000 }
gfCNCPoint2[13073] = {X 397.1171, Y 87.3474, Z -3.0000, A 0.000, B 0.000, C 0.000 }
gfCNCPoint2[13074] = {X 416.3162, Y 75.0513, Z -3.0000, A 0.000, B 0.000, C 0.000 }
gfCNCPoint2[13075] = {X 401.7935, Y 69.3532, Z -3.0000, A 0.000, B 0.000, C 0.000 }
gfCNCPoint2[13076] = {X 400.6813, Y 68.9834, Z -3.0000, A 0.000, B 0.000, C 0.000 }
gfCNCPoint2[13077] = {X 399.5358, Y 68.7355, Z -3.0000, A 0.000, B 0.000, C 0.000 }
gfCNCPoint2[13078] = {X 398.3702, Y 68.6122, Z -3.0000, A 0.000, B 0.000, C 0.000 }
gfCNCPoint2[13079] = {X 397.6035, Y 68.5669, Z -3.0000, A 0.000, B 0.000, C 0.000 }
gfCNCPoint2[13080] = {X 396.8428, Y 68.4609, Z -3.0000, A 0.000, B 0.000, C 0.000 }
gfCNCPoint2[13081] = {X 395.3924, Y 68.0819, Z -3.0000, A 0.000, B 0.000, C 0.000 }
gfCNCPoint2[13082] = {X 394.0179, Y 67.4835, Z -3.0000, A 0.000, B 0.000, C 0.000 }
gfCNCPoint2[13083] = {X 394.0174, Y 73.4813, Z -3.0000, A 0.000, B 0.000, C 0.000 }
gfCNCPoint2[13084] = {X 391.6174, Y 73.4811, Z -3.0000, A 0.000, B 0.000, C 0.000 }
gfCNCPoint2[13085] = {X 391.6163, Y 84.6052, Z -3.0000, A 0.000, B 0.000, C 0.000 }
gfCNCPoint2[13086] = {X 391.5803, Y 86.0256, Z -3.0000, A 0.000, B 0.000, C 0.000 }
gfCNCPoint2[13087] = {X 391.4526, Y 87.4406, Z -3.0000, A 0.000, B 0.000, C 0.000 }
gfCNCPoint2[13088] = {X 391.2282, Y 88.8724, Z -3.0000, A 0.000, B 0.000, C 0.000 }
gfCNCPoint2[13089] = {X 390.9099, Y 90.2862, Z -3.0000, A 0.000, B 0.000, C 0.000 }
gfCNCPoint2[13090] = {X 390.3338, Y 92.0500, Z -3.0000, A 0.000, B 0.000, C 0.000 }
gfCNCPoint2[13091] = {X 389.5424, Y 93.7283, Z -3.0000, A 0.000, B 0.000, C 0.000 }
gfCNCPoint2[13092] = {X 388.5481, Y 95.2950, Z -3.0000, A 0.000, B 0.000, C 0.000 }
gfCNCPoint2[13093] = {X 389.3446, Y 95.2950, Z -3.0000, A 0.000, B 0.000, C 0.000 }
gfCNCPoint2[13094] = {X 389.7639, Y 94.0857, Z -3.0000, A 0.000, B 0.000, C 0.000 }
gfCNCPoint2[13095] = {X 390.3885, Y 92.9686, Z -3.0000, A 0.000, B 0.000, C 0.000 }
gfCNCPoint2[13096] = {X 391.1990, Y 91.9781, Z -3.0000, A 0.000, B 0.000, C 0.000 }
gfCNCPoint2[13097] = {X 392.1705, Y 91.1448, Z -3.0000, A 0.000, B 0.000, C 0.000 }
gfCNCPoint2[13098] = {X 393.2729, Y 90.4946, Z -3.0000, A 0.000, B 0.000, C 0.000 }
gfCNCPoint2[13099] = {X 394.4721, Y 90.0475, Z -3.0000, A 0.000, B 0.000, C 0.000 }
gfCNCPoint2[13100] = {X 395.4058, Y 89.8550, Z -3.0000, A 0.000, B 0.000, C 0.000 }
gfCNCPoint2[13101] = {X 396.3567, Y 89.7861, Z -3.0000, A 0.000, B 0.000, C 0.000 }
gfCNCPoint2[13102] = {X 397.1493, Y 89.7490, Z -3.0000, A 0.000, B 0.000, C 0.000 }
gfCNCPoint2[13103] = {X 397.9389, Y 89.6711, Z -3.0000, A 0.000, B 0.000, C 0.000 }
gfCNCPoint2[13104] = {X 421.5719, Y 74.5353, Z -3.0000, A 0.000, B 0.000, C 0.000 }
gfCNCPoint2[13105] = {X 402.6722, Y 67.1198, Z -3.0000, A 0.000, B 0.000, C 0.000 }
gfCNCPoint2[13106] = {X 401.3007, Y 66.6647, Z -3.0000, A 0.000, B 0.000, C 0.000 }
gfCNCPoint2[13107] = {X 399.8880, Y 66.3613, Z -3.0000, A 0.000, B 0.000, C 0.000 }
gfCNCPoint2[13108] = {X 398.4506, Y 66.2133, Z -3.0000, A 0.000, B 0.000, C 0.000 }
gfCNCPoint2[13109] = {X 397.3060, Y 66.1056, Z -3.0000, A 0.000, B 0.000, C 0.000 }
gfCNCPoint2[13110] = {X 396.1926, Y 65.8192, Z -3.0000, A 0.000, B 0.000, C 0.000 }
gfCNCPoint2[13111] = {X 395.1382, Y 65.3610, Z -3.0000, A 0.000, B 0.000, C 0.000 }
gfCNCPoint2[13112] = {X 394.1691, Y 64.7425, Z -3.0000, A 0.000, B 0.000, C 0.000 }
gfCNCPoint2[13113] = {X 393.3094, Y 63.9792, Z -3.0000, A 0.000, B 0.000, C 0.000 }
gfCNCPoint2[13114] = {X 392.5120, Y 64.6965, Z -3.0000, A 0.000, B 0.000, C 0.000 }
gfCNCPoint2[13115] = {X 391.6181, Y 65.2893, Z -3.0000, A 0.000, B 0.000, C 0.000 }
gfCNCPoint2[13116] = {X 391.6174, Y 73.4811, Z -3.0000, A 0.000, B 0.000, C 0.000 }
gfCNCPoint2[13117] = {X 389.2174, Y 73.4809, Z -3.0000, A 0.000, B 0.000, C 0.000 }
gfCNCPoint2[13118] = {X 389.2163, Y 84.6138, Z -3.0000, A 0.000, B 0.000, C 0.000 }
gfCNCPoint2[13119] = {X 389.1545, Y 86.3199, Z -3.0000, A 0.000, B 0.000, C 0.000 }
gfCNCPoint2[13120] = {X 388.9442, Y 88.0141, Z -3.0000, A 0.000, B 0.000, C 0.000 }
gfCNCPoint2[13121] = {X 388.5868, Y 89.6834, Z -3.0000, A 0.000, B 0.000, C 0.000 }
gfCNCPoint2[13122] = {X 388.1037, Y 91.1630, Z -3.0000, A 0.000, B 0.000, C 0.000 }
gfCNCPoint2[13123] = {X 387.4400, Y 92.5708, Z -3.0000, A 0.000, B 0.000, C 0.000 }
gfCNCPoint2[13124] = {X 386.6060, Y 93.8849, Z -3.0000, A 0.000, B 0.000, C 0.000 }
gfCNCPoint2[13125] = {X 385.8737, Y 94.7997, Z -3.0000, A 0.000, B 0.000, C 0.000 }
gfCNCPoint2[13126] = {X 385.0588, Y 95.6417, Z -3.0000, A 0.000, B 0.000, C 0.000 }
gfCNCPoint2[13127] = {X 383.7987, Y 96.7249, Z -3.0000, A 0.000, B 0.000, C 0.000 }
gfCNCPoint2[13128] = {X 382.4496, Y 97.6950, Z -3.0000, A 0.000, B 0.000, C 0.000 }
gfCNCPoint2[13129] = {X 382.1865, Y 97.2935, Z -3.0000, A 0.000, B 0.000, C 0.000 }
gfCNCPoint2[13130] = {X 381.0194, Y 97.9989, Z -3.0000, A 0.000, B 0.000, C 0.000 }
gfCNCPoint2[13131] = {X 379.8040, Y 98.6175, Z -3.0000, A 0.000, B 0.000, C 0.000 }
gfCNCPoint2[13132] = {X 377.5271, Y 99.5760, Z -3.0000, A 0.000, B 0.000, C 0.000 }
gfCNCPoint2[13133] = {X 375.1871, Y 100.3682, Z -3.0000, A 0.000, B 0.000, C 0.000 }
gfCNCPoint2[13134] = {X 372.7962, Y 100.9900, Z -3.0000, A 0.000, B 0.000, C 0.000 }
gfCNCPoint2[13135] = {X 368.9811, Y 101.7281, Z -3.0000, A 0.000, B 0.000, C 0.000 }
gfCNCPoint2[13136] = {X 365.1349, Y 102.2819, Z -3.0000, A 0.000, B 0.000, C 0.000 }
gfCNCPoint2[13137] = {X 361.2665, Y 102.6502, Z -3.0000, A 0.000, B 0.000, C 0.000 }
gfCNCPoint2[13138] = {X 355.1239, Y 102.9835, Z -3.0000, A 0.000, B 0.000, C 0.000 }
gfCNCPoint2[13139] = {X 348.9736, Y 103.1120, Z -3.0000, A 0.000, B 0.000, C 0.000 }
gfCNCPoint2[13140] = {X 342.8225, Y 103.0356, Z -3.0000, A 0.000, B 0.000, C 0.000 }
gfCNCPoint2[13141] = {X 336.6773, Y 102.7543, Z -3.0000, A 0.000, B 0.000, C 0.000 }
gfCNCPoint2[13142] = {X 333.1845, Y 102.4780, Z -3.0000, A 0.000, B 0.000, C 0.000 }
gfCNCPoint2[13143] = {X 329.7052, Y 102.0647, Z -3.0000, A 0.000, B 0.000, C 0.000 }
gfCNCPoint2[13144] = {X 326.2448, Y 101.5151, Z -3.0000, A 0.000, B 0.000, C 0.000 }
gfCNCPoint2[13145] = {X 323.3898, Y 100.9089, Z -3.0000, A 0.000, B 0.000, C 0.000 }
gfCNCPoint2[13146] = {X 320.5870, Y 100.0944, Z -3.0000, A 0.000, B 0.000, C 0.000 }
gfCNCPoint2[13147] = {X 317.8518, Y 99.0759, Z -3.0000, A 0.000, B 0.000, C 0.000 }
gfCNCPoint2[13148] = {X 316.3332, Y 98.3748, Z -3.0000, A 0.000, B 0.000, C 0.000 }
gfCNCPoint2[13149] = {X 314.8783, Y 97.5496, Z -3.0000, A 0.000, B 0.000, C 0.000 }
gfCNCPoint2[13150] = {X 313.4973, Y 96.6059, Z -3.0000, A 0.000, B 0.000, C 0.000 }
gfCNCPoint2[13151] = {X 312.1998, Y 95.5504, Z -3.0000, A 0.000, B 0.000, C 0.000 }
gfCNCPoint2[13152] = {X 311.1892, Y 94.5454, Z -3.0000, A 0.000, B 0.000, C 0.000 }
gfCNCPoint2[13153] = {X 310.3050, Y 93.4275, Z -3.0000, A 0.000, B 0.000, C 0.000 }
gfCNCPoint2[13154] = {X 309.5597, Y 92.2126, Z -3.0000, A 0.000, B 0.000, C 0.000 }
gfCNCPoint2[13155] = {X 308.9638, Y 90.9179, Z -3.0000, A 0.000, B 0.000, C 0.000 }
gfCNCPoint2[13156] = {X 308.5257, Y 89.5616, Z -3.0000, A 0.000, B 0.000, C 0.000 }
gfCNCPoint2[13157] = {X 308.1809, Y 87.9321, Z -3.0000, A 0.000, B 0.000, C 0.000 }
gfCNCPoint2[13158] = {X 307.9772, Y 86.2789, Z -3.0000, A 0.000, B 0.000, C 0.000 }
gfCNCPoint2[13159] = {X 307.9160, Y 84.6144, Z -3.0000, A 0.000, B 0.000, C 0.000 }
gfCNCPoint2[13160] = {X 307.9173, Y 83.2309, Z -3.0000, A 0.000, B 0.000, C 0.000 }
gfCNCPoint2[13161] = {X 307.9173, Y 63.2814, Z -3.0000, A 0.000, B 0.000, C 0.000 }
gfCNCPoint2[13162] = {X 307.0578, Y 63.0564, Z -3.0000, A 0.000, B 0.000, C 0.000 }
gfCNCPoint2[13163] = {X 306.2610, Y 62.6633, Z -3.0000, A 0.000, B 0.000, C 0.000 }
gfCNCPoint2[13164] = {X 305.5595, Y 62.1181, Z -3.0000, A 0.000, B 0.000, C 0.000 }
gfCNCPoint2[13165] = {X 304.9817, Y 61.4431, Z -3.0000, A 0.000, B 0.000, C 0.000 }
gfCNCPoint2[13166] = {X 304.5514, Y 60.6659, Z -3.0000, A 0.000, B 0.000, C 0.000 }
gfCNCPoint2[13167] = {X 304.2859, Y 59.8180, Z -3.0000, A 0.000, B 0.000, C 0.000 }
gfCNCPoint2[13168] = {X 304.1962, Y 58.9340, Z -3.0000, A 0.000, B 0.000, C 0.000 }
gfCNCPoint2[13169] = {X 304.1962, Y 58.0000, Z -3.0000, A 0.000, B 0.000, C 0.000 }
gfCNCPoint2[13170] = {X 304.3065, Y 57.0209, Z -3.0000, A 0.000, B 0.000, C 0.000 }
gfCNCPoint2[13171] = {X 304.6320, Y 56.0909, Z -3.0000, A 0.000, B 0.000, C 0.000 }
gfCNCPoint2[13172] = {X 305.1562, Y 55.2566, Z -3.0000, A 0.000, B 0.000, C 0.000 }
gfCNCPoint2[13173] = {X 305.8529, Y 54.5599, Z -3.0000, A 0.000, B 0.000, C 0.000 }
gfCNCPoint2[13174] = {X 306.6871, Y 54.0357, Z -3.0000, A 0.000, B 0.000, C 0.000 }
gfCNCPoint2[13175] = {X 307.6171, Y 53.7103, Z -3.0000, A 0.000, B 0.000, C 0.000 }
gfCNCPoint2[13176] = {X 308.5962, Y 53.6000, Z -3.0000, A 0.000, B 0.000, C 0.000 }
gfCNCPoint2[13177] = {X 324.3107, Y 53.6000, Z -3.0000, A 0.000, B 0.000, C 0.000 }
gfCNCPoint2[13178] = {X 325.2898, Y 53.7103, Z -3.0000, A 0.000, B 0.000, C 0.000 }
gfCNCPoint2[13179] = {X 326.2198, Y 54.0357, Z -3.0000, A 0.000, B 0.000, C 0.000 }
gfCNCPoint2[13180] = {X 327.0540, Y 54.5599, Z -3.0000, A 0.000, B 0.000, C 0.000 }
gfCNCPoint2[13181] = {X 327.7507, Y 55.2566, Z -3.0000, A 0.000, B 0.000, C 0.000 }
gfCNCPoint2[13182] = {X 328.2750, Y 56.0909, Z -3.0000, A 0.000, B 0.000, C 0.000 }
gfCNCPoint2[13183] = {X 328.6004, Y 57.0209, Z -3.0000, A 0.000, B 0.000, C 0.000 }
gfCNCPoint2[13184] = {X 328.7107, Y 58.0000, Z -3.0000, A 0.000, B 0.000, C 0.000 }
gfCNCPoint2[13185] = {X 328.7107, Y 58.9365, Z -3.0000, A 0.000, B 0.000, C 0.000 }
gfCNCPoint2[13186] = {X 328.6166, Y 59.8191, Z -3.0000, A 0.000, B 0.000, C 0.000 }
gfCNCPoint2[13187] = {X 328.3489, Y 60.6654, Z -3.0000, A 0.000, B 0.000, C 0.000 }
gfCNCPoint2[13188] = {X 327.9181, Y 61.4415, Z -3.0000, A 0.000, B 0.000, C 0.000 }
gfCNCPoint2[13189] = {X 327.3415, Y 62.1163, Z -3.0000, A 0.000, B 0.000, C 0.000 }
gfCNCPoint2[13190] = {X 326.6422, Y 62.6630, Z -3.0000, A 0.000, B 0.000, C 0.000 }
gfCNCPoint2[13191] = {X 325.8482, Y 63.0596, Z -3.0000, A 0.000, B 0.000, C 0.000 }
gfCNCPoint2[13192] = {X 324.9911, Y 63.2904, Z -3.0000, A 0.000, B 0.000, C 0.000 }
gfCNCPoint2[13193] = {X 324.9926, Y 83.2292, Z -3.0000, A 0.000, B 0.000, C 0.000 }
gfCNCPoint2[13194] = {X 325.0061, Y 84.6145, Z -3.0000, A 0.000, B 0.000, C 0.000 }
gfCNCPoint2[13195] = {X 325.0819, Y 85.8326, Z -3.0000, A 0.000, B 0.000, C 0.000 }
gfCNCPoint2[13196] = {X 325.3001, Y 87.0334, Z -3.0000, A 0.000, B 0.000, C 0.000 }
gfCNCPoint2[13197] = {X 325.5331, Y 87.2842, Z -3.0000, A 0.000, B 0.000, C 0.000 }
gfCNCPoint2[13198] = {X 325.8186, Y 87.4730, Z -3.0000, A 0.000, B 0.000, C 0.000 }
gfCNCPoint2[13199] = {X 326.2610, Y 87.7228, Z -3.0000, A 0.000, B 0.000, C 0.000 }
gfCNCPoint2[13200] = {X 327.6906, Y 88.3165, Z -3.0000, A 0.000, B 0.000, C 0.000 }
gfCNCPoint2[13201] = {X 329.1769, Y 88.7492, Z -3.0000, A 0.000, B 0.000, C 0.000 }
gfCNCPoint2[13202] = {X 332.2475, Y 89.3639, Z -3.0000, A 0.000, B 0.000, C 0.000 }
gfCNCPoint2[13203] = {X 335.3543, Y 89.7557, Z -3.0000, A 0.000, B 0.000, C 0.000 }
gfCNCPoint2[13204] = {X 339.4910, Y 90.0761, Z -3.0000, A 0.000, B 0.000, C 0.000 }
gfCNCPoint2[13205] = {X 343.6362, Y 90.2556, Z -3.0000, A 0.000, B 0.000, C 0.000 }
gfCNCPoint2[13206] = {X 347.7851, Y 90.2940, Z -3.0000, A 0.000, B 0.000, C 0.000 }
gfCNCPoint2[13207] = {X 352.1632, Y 90.2556, Z -3.0000, A 0.000, B 0.000, C 0.000 }
gfCNCPoint2[13208] = {X 356.5371, Y 90.0598, Z -3.0000, A 0.000, B 0.000, C 0.000 }
gfCNCPoint2[13209] = {X 360.9012, Y 89.7069, Z -3.0000, A 0.000, B 0.000, C 0.000 }
gfCNCPoint2[13210] = {X 363.2108, Y 89.4196, Z -3.0000, A 0.000, B 0.000, C 0.000 }
gfCNCPoint2[13211] = {X 365.4989, Y 88.9939, Z -3.0000, A 0.000, B 0.000, C 0.000 }
gfCNCPoint2[13212] = {X 367.7574, Y 88.4315, Z -3.0000, A 0.000, B 0.000, C 0.000 }
gfCNCPoint2[13213] = {X 368.6803, Y 88.1211, Z -3.0000, A 0.000, B 0.000, C 0.000 }
gfCNCPoint2[13214] = {X 369.5626, Y 87.7091, Z -3.0000, A 0.000, B 0.000, C 0.000 }
gfCNCPoint2[13215] = {X 370.3932, Y 87.2009, Z -3.0000, A 0.000, B 0.000, C 0.000 }
gfCNCPoint2[13216] = {X 370.5211, Y 87.0678, Z -3.0000, A 0.000, B 0.000, C 0.000 }
gfCNCPoint2[13217] = {X 370.5870, Y 86.8954, Z -3.0000, A 0.000, B 0.000, C 0.000 }
gfCNCPoint2[13218] = {X 370.7773, Y 85.3669, Z -3.0000, A 0.000, B 0.000, C 0.000 }
gfCNCPoint2[13219] = {X 370.8408, Y 83.8280, Z -3.0000, A 0.000, B 0.000, C 0.000 }
gfCNCPoint2[13220] = {X 370.8391, Y 63.2812, Z -3.0000, A 0.000, B 0.000, C 0.000 }
gfCNCPoint2[13221] = {X 369.9799, Y 63.0560, Z -3.0000, A 0.000, B 0.000, C 0.000 }
gfCNCPoint2[13222] = {X 369.1833, Y 62.6628, Z -3.0000, A 0.000, B 0.000, C 0.000 }
gfCNCPoint2[13223] = {X 368.4820, Y 62.1176, Z -3.0000, A 0.000, B 0.000, C 0.000 }
gfCNCPoint2[13224] = {X 367.9045, Y 61.4427, Z -3.0000, A 0.000, B 0.000, C 0.000 }
gfCNCPoint2[13225] = {X 367.4743, Y 60.6655, Z -3.0000, A 0.000, B 0.000, C 0.000 }
gfCNCPoint2[13226] = {X 367.2089, Y 59.8178, Z -3.0000, A 0.000, B 0.000, C 0.000 }
gfCNCPoint2[13227] = {X 367.1193, Y 58.9340, Z -3.0000, A 0.000, B 0.000, C 0.000 }
gfCNCPoint2[13228] = {X 367.1193, Y 58.0000, Z -3.0000, A 0.000, B 0.000, C 0.000 }
gfCNCPoint2[13229] = {X 367.2296, Y 57.0209, Z -3.0000, A 0.000, B 0.000, C 0.000 }
gfCNCPoint2[13230] = {X 367.5550, Y 56.0909, Z -3.0000, A 0.000, B 0.000, C 0.000 }
gfCNCPoint2[13231] = {X 368.0792, Y 55.2566, Z -3.0000, A 0.000, B 0.000, C 0.000 }
gfCNCPoint2[13232] = {X 368.7759, Y 54.5599, Z -3.0000, A 0.000, B 0.000, C 0.000 }
gfCNCPoint2[13233] = {X 369.6102, Y 54.0357, Z -3.0000, A 0.000, B 0.000, C 0.000 }
gfCNCPoint2[13234] = {X 370.5402, Y 53.7103, Z -3.0000, A 0.000, B 0.000, C 0.000 }
gfCNCPoint2[13235] = {X 371.5193, Y 53.6000, Z -3.0000, A 0.000, B 0.000, C 0.000 }
gfCNCPoint2[13236] = {X 388.0597, Y 53.6000, Z -3.0000, A 0.000, B 0.000, C 0.000 }
gfCNCPoint2[13237] = {X 389.0388, Y 53.7103, Z -3.0000, A 0.000, B 0.000, C 0.000 }
gfCNCPoint2[13238] = {X 389.9688, Y 54.0357, Z -3.0000, A 0.000, B 0.000, C 0.000 }
gfCNCPoint2[13239] = {X 390.8030, Y 54.5599, Z -3.0000, A 0.000, B 0.000, C 0.000 }
gfCNCPoint2[13240] = {X 391.4997, Y 55.2566, Z -3.0000, A 0.000, B 0.000, C 0.000 }
gfCNCPoint2[13241] = {X 392.0239, Y 56.0909, Z -3.0000, A 0.000, B 0.000, C 0.000 }
gfCNCPoint2[13242] = {X 392.3494, Y 57.0209, Z -3.0000, A 0.000, B 0.000, C 0.000 }
gfCNCPoint2[13243] = {X 392.4597, Y 58.0000, Z -3.0000, A 0.000, B 0.000, C 0.000 }
gfCNCPoint2[13244] = {X 392.4595, Y 58.9704, Z -3.0000, A 0.000, B 0.000, C 0.000 }
gfCNCPoint2[13245] = {X 392.3382, Y 59.9609, Z -3.0000, A 0.000, B 0.000, C 0.000 }
gfCNCPoint2[13246] = {X 391.9968, Y 60.8986, Z -3.0000, A 0.000, B 0.000, C 0.000 }
gfCNCPoint2[13247] = {X 391.5530, Y 61.6099, Z -3.0000, A 0.000, B 0.000, C 0.000 }
